Fanuc TP program (LS listing): hs_ov_h80_gutr1.ls

/PROG  hs_ov_h80_gutr1
/ATTR
COMMENT	= "19-03-05 13:35:50";
PROG_SIZE	= 0;
DEFAULT_GROUP	= 1, *, *, *, *;
/APPL
    ARC Welding Equipment: 1, *, *, *, *;
/MN
   1:  CALL HOME_ALL;
   1:  UFRAME_NUM = 1;
   1:  UTOOL_NUM = 3;
   1:  COL GUARD ADJUST 150;
   1:  PR[91] = PR[90];
   1:  PR[91,1] = PR[90,1] + -0.906;
   1:  PR[91,2] = PR[90,2] + 14.621;
   1:  PR[91,3] = PR[90,3] + 36.595;
   1:  PR[92] = PR[91];
   1:  PR[92,3] = PR[92,3] + 50;
   1:J PR[92] 10% FINE;
   1:L PR[91] R[100]mm/sec CNT100;
   1:  CALL LASER_DRAHT_START;
   1:  PR[91,1] = PR[90,1] + -1.737;
   1:  PR[91,2] = PR[90,2] + 15.006;
   1:L PR[91] R[100]mm/sec CNT100;
   1:  PR[91,1] = PR[90,1] + -2.132;
   1:  PR[91,2] = PR[90,2] + 15.132;
   1:L PR[91] R[100]mm/sec CNT100;
   1:  PR[91,1] = PR[90,1] + -6.402;
   1:  PR[91,2] = PR[90,2] + 17.485;
   1:L PR[91] R[100]mm/sec CNT100;
   1:  PR[91,1] = PR[90,1] + -10.845;
   1:  PR[91,2] = PR[90,2] + 18.832;
   1:L PR[91] R[100]mm/sec CNT100;
   1:  PR[91,1] = PR[90,1] + -10.901;
   1:  PR[91,2] = PR[90,2] + 18.841;
   1:L PR[91] R[100]mm/sec CNT100;
   1:  PR[91,1] = PR[90,1] + -15.199;
   1:  PR[91,2] = PR[90,2] + 19.185;
   1:L PR[91] R[100]mm/sec CNT100;
   1:  PR[91,1] = PR[90,1] + -15.522;
   1:  PR[91,2] = PR[90,2] + 19.196;
   1:L PR[91] R[100]mm/sec CNT100;
   1:  PR[91,1] = PR[90,1] + -15.935;
   1:  PR[91,2] = PR[90,2] + 19.155;
   1:L PR[91] R[100]mm/sec CNT100;
   1:  PR[91,1] = PR[90,1] + -19.834;
   1:  PR[91,2] = PR[90,2] + 18.637;
   1:L PR[91] R[100]mm/sec CNT100;
   1:  PR[91,1] = PR[90,1] + -20.377;
   1:  PR[91,2] = PR[90,2] + 18.508;
   1:L PR[91] R[100]mm/sec CNT100;
   1:  PR[91,1] = PR[90,1] + -21.139;
   1:  PR[91,2] = PR[90,2] + 18.219;
   1:L PR[91] R[100]mm/sec CNT100;
   1:  PR[91,1] = PR[90,1] + -24.417;
   1:  PR[91,2] = PR[90,2] + 17.039;
   1:L PR[91] R[100]mm/sec CNT100;
   1:  PR[91,1] = PR[90,1] + -25.209;
   1:  PR[91,2] = PR[90,2] + 16.607;
   1:L PR[91] R[100]mm/sec CNT100;
   1:  PR[91,1] = PR[90,1] + -27.740;
   1:  PR[91,2] = PR[90,2] + 15.030;
   1:L PR[91] R[100]mm/sec CNT100;
   1:  PR[91,1] = PR[90,1] + -28.583;
   1:  PR[91,2] = PR[90,2] + 14.408;
   1:L PR[91] R[100]mm/sec CNT100;
   1:  PR[91,1] = PR[90,1] + -31.305;
   1:  PR[91,2] = PR[90,2] + 11.747;
   1:L PR[91] R[100]mm/sec CNT100;
   1:  PR[91,1] = PR[90,1] + -32.081;
   1:  PR[91,2] = PR[90,2] + 10.737;
   1:L PR[91] R[100]mm/sec CNT100;
   1:  PR[91,1] = PR[90,1] + -33.285;
   1:  PR[91,2] = PR[90,2] + 8.860;
   1:L PR[91] R[100]mm/sec CNT100;
   1:  PR[91,1] = PR[90,1] + -33.988;
   1:  PR[91,2] = PR[90,2] + 7.608;
   1:L PR[91] R[100]mm/sec CNT100;
   1:  PR[91,1] = PR[90,1] + -34.555;
   1:  PR[91,2] = PR[90,2] + 6.149;
   1:L PR[91] R[100]mm/sec CNT100;
   1:  PR[91,1] = PR[90,1] + -35.218;
   1:  PR[91,2] = PR[90,2] + 4.337;
   1:L PR[91] R[100]mm/sec CNT100;
   1:  PR[91,1] = PR[90,1] + -35.516;
   1:  PR[91,2] = PR[90,2] + 3.007;
   1:L PR[91] R[100]mm/sec CNT100;
   1:  PR[91,1] = PR[90,1] + -35.629;
   1:  PR[91,2] = PR[90,2] + 1.384;
   1:L PR[91] R[100]mm/sec CNT100;
   1:  PR[91,1] = PR[90,1] + -35.844;
   1:  PR[91,2] = PR[90,2] + -0.479;
   1:L PR[91] R[100]mm/sec CNT100;
   1:  PR[91,1] = PR[90,1] + -35.742;
   1:  PR[91,2] = PR[90,2] + -1.958;
   1:L PR[91] R[100]mm/sec CNT100;
   1:  PR[91,1] = PR[90,1] + -35.528;
   1:  PR[91,2] = PR[90,2] + -3.801;
   1:L PR[91] R[100]mm/sec CNT100;
   1:  PR[91,1] = PR[90,1] + -35.224;
   1:  PR[91,2] = PR[90,2] + -5.160;
   1:L PR[91] R[100]mm/sec CNT100;
   1:  PR[91,1] = PR[90,1] + -34.654;
   1:  PR[91,2] = PR[90,2] + -6.622;
   1:L PR[91] R[100]mm/sec CNT100;
   1:  PR[91,1] = PR[90,1] + -33.976;
   1:  PR[91,2] = PR[90,2] + -8.476;
   1:L PR[91] R[100]mm/sec CNT100;
   1:  PR[91,1] = PR[90,1] + -33.285;
   1:  PR[91,2] = PR[90,2] + -9.707;
   1:L PR[91] R[100]mm/sec CNT100;
   1:  PR[91,1] = PR[90,1] + -32.081;
   1:  PR[91,2] = PR[90,2] + -11.584;
   1:L PR[91] R[100]mm/sec CNT100;
   1:  PR[91,1] = PR[90,1] + -31.305;
   1:  PR[91,2] = PR[90,2] + -12.594;
   1:L PR[91] R[100]mm/sec CNT100;
   1:  PR[91,1] = PR[90,1] + -28.583;
   1:  PR[91,2] = PR[90,2] + -15.255;
   1:L PR[91] R[100]mm/sec CNT100;
   1:  PR[91,1] = PR[90,1] + -27.740;
   1:  PR[91,2] = PR[90,2] + -15.877;
   1:L PR[91] R[100]mm/sec CNT100;
   1:  PR[91,1] = PR[90,1] + -25.208;
   1:  PR[91,2] = PR[90,2] + -17.454;
   1:L PR[91] R[100]mm/sec CNT100;
   1:  PR[91,1] = PR[90,1] + -24.396;
   1:  PR[91,2] = PR[90,2] + -17.898;
   1:L PR[91] R[100]mm/sec CNT100;
   1:  PR[91,1] = PR[90,1] + -23.616;
   1:  PR[91,2] = PR[90,2] + -18.195;
   1:L PR[91] R[100]mm/sec CNT100;
   1:  PR[91,1] = PR[90,1] + -20.398;
   1:  PR[91,2] = PR[90,2] + -19.351;
   1:L PR[91] R[100]mm/sec CNT100;
   1:  PR[91,1] = PR[90,1] + -19.877;
   1:  PR[91,2] = PR[90,2] + -19.474;
   1:L PR[91] R[100]mm/sec CNT100;
   1:  PR[91,1] = PR[90,1] + -19.263;
   1:  PR[91,2] = PR[90,2] + -19.533;
   1:L PR[91] R[100]mm/sec CNT100;
   1:  PR[91,1] = PR[90,1] + -15.479;
   1:  PR[91,2] = PR[90,2] + -20.042;
   1:L PR[91] R[100]mm/sec CNT100;
   1:  PR[91,1] = PR[90,1] + -15.199;
   1:  PR[91,2] = PR[90,2] + -20.033;
   1:L PR[91] R[100]mm/sec CNT100;
   1:  PR[91,1] = PR[90,1] + -10.901;
   1:  PR[91,2] = PR[90,2] + -19.688;
   1:L PR[91] R[100]mm/sec CNT100;
   1:  PR[91,1] = PR[90,1] + -10.845;
   1:  PR[91,2] = PR[90,2] + -19.679;
   1:L PR[91] R[100]mm/sec CNT100;
   1:  PR[91,1] = PR[90,1] + -6.401;
   1:  PR[91,2] = PR[90,2] + -18.332;
   1:L PR[91] R[100]mm/sec CNT100;
   1:  PR[91,1] = PR[90,1] + -2.136;
   1:  PR[91,2] = PR[90,2] + -15.981;
   1:L PR[91] R[100]mm/sec CNT100;
   1:  PR[91,1] = PR[90,1] + -1.638;
   1:  PR[91,2] = PR[90,2] + -15.821;
   1:L PR[91] R[100]mm/sec CNT100;
   1:  PR[91,1] = PR[90,1] + -1.622;
   1:  PR[91,2] = PR[90,2] + -15.815;
   1:L PR[91] R[100]mm/sec CNT100;
   1:  PR[91,1] = PR[90,1] + -0.788;
   1:  PR[91,2] = PR[90,2] + -15.263;
   1:L PR[91] R[100]mm/sec CNT100;
   1:  PR[91,1] = PR[90,1] + 0.384;
   1:  PR[91,2] = PR[90,2] + -15.590;
   1:L PR[91] R[100]mm/sec CNT100;
   1:  PR[91,1] = PR[90,1] + 1.398;
   1:  PR[91,2] = PR[90,2] + -15.747;
   1:L PR[91] R[100]mm/sec CNT100;
   1:  PR[91,1] = PR[90,1] + 1.978;
   1:  PR[91,2] = PR[90,2] + -16.161;
   1:L PR[91] R[100]mm/sec CNT100;
   1:  PR[91,1] = PR[90,1] + 5.916;
   1:  PR[91,2] = PR[90,2] + -18.330;
   1:L PR[91] R[100]mm/sec CNT100;
   1:  PR[91,1] = PR[90,1] + 10.362;
   1:  PR[91,2] = PR[90,2] + -19.678;
   1:L PR[91] R[100]mm/sec CNT100;
   1:  PR[91,1] = PR[90,1] + 10.418;
   1:  PR[91,2] = PR[90,2] + -19.687;
   1:L PR[91] R[100]mm/sec CNT100;
   1:  PR[91,1] = PR[90,1] + 14.716;
   1:  PR[91,2] = PR[90,2] + -20.033;
   1:L PR[91] R[100]mm/sec CNT100;
   1:  PR[91,1] = PR[90,1] + 15.037;
   1:  PR[91,2] = PR[90,2] + -20.044;
   1:L PR[91] R[100]mm/sec CNT100;
   1:  PR[91,1] = PR[90,1] + 15.446;
   1:  PR[91,2] = PR[90,2] + -20.004;
   1:L PR[91] R[100]mm/sec CNT100;
   1:  PR[91,1] = PR[90,1] + 19.345;
   1:  PR[91,2] = PR[90,2] + -19.485;
   1:L PR[91] R[100]mm/sec CNT100;
   1:  PR[91,1] = PR[90,1] + 19.888;
   1:  PR[91,2] = PR[90,2] + -19.357;
   1:L PR[91] R[100]mm/sec CNT100;
   1:  PR[91,1] = PR[90,1] + 20.651;
   1:  PR[91,2] = PR[90,2] + -19.069;
   1:L PR[91] R[100]mm/sec CNT100;
   1:  PR[91,1] = PR[90,1] + 23.931;
   1:  PR[91,2] = PR[90,2] + -17.890;
   1:L PR[91] R[100]mm/sec CNT100;
   1:  PR[91,1] = PR[90,1] + 24.719;
   1:  PR[91,2] = PR[90,2] + -17.462;
   1:L PR[91] R[100]mm/sec CNT100;
   1:  PR[91,1] = PR[90,1] + 27.251;
   1:  PR[91,2] = PR[90,2] + -15.887;
   1:L PR[91] R[100]mm/sec CNT100;
   1:  PR[91,1] = PR[90,1] + 28.082;
   1:  PR[91,2] = PR[90,2] + -15.277;
   1:L PR[91] R[100]mm/sec CNT100;
   1:  PR[91,1] = PR[90,1] + 30.802;
   1:  PR[91,2] = PR[90,2] + -12.615;
   1:L PR[91] R[100]mm/sec CNT100;
   1:  PR[91,1] = PR[90,1] + 31.587;
   1:  PR[91,2] = PR[90,2] + -11.595;
   1:L PR[91] R[100]mm/sec CNT100;
   1:  PR[91,1] = PR[90,1] + 32.794;
   1:  PR[91,2] = PR[90,2] + -9.717;
   1:L PR[91] R[100]mm/sec CNT100;
   1:  PR[91,1] = PR[90,1] + 33.504;
   1:  PR[91,2] = PR[90,2] + -8.463;
   1:L PR[91] R[100]mm/sec CNT100;
   1:  PR[91,1] = PR[90,1] + 34.067;
   1:  PR[91,2] = PR[90,2] + -7.036;
   1:L PR[91] R[100]mm/sec CNT100;
   1:  PR[91,1] = PR[90,1] + 34.729;
   1:  PR[91,2] = PR[90,2] + -5.233;
   1:L PR[91] R[100]mm/sec CNT100;
   1:  PR[91,1] = PR[90,1] + 35.030;
   1:  PR[91,2] = PR[90,2] + -3.913;
   1:L PR[91] R[100]mm/sec CNT100;
   1:  PR[91,1] = PR[90,1] + 35.150;
   1:  PR[91,2] = PR[90,2] + -2.237;
   1:L PR[91] R[100]mm/sec CNT100;
   1:  PR[91,1] = PR[90,1] + 35.364;
   1:  PR[91,2] = PR[90,2] + -0.371;
   1:L PR[91] R[100]mm/sec CNT100;
   1:  PR[91,1] = PR[90,1] + 35.255;
   1:  PR[91,2] = PR[90,2] + 1.165;
   1:L PR[91] R[100]mm/sec CNT100;
   1:  PR[91,1] = PR[90,1] + 35.042;
   1:  PR[91,2] = PR[90,2] + 3.015;
   1:L PR[91] R[100]mm/sec CNT100;
   1:  PR[91,1] = PR[90,1] + 34.736;
   1:  PR[91,2] = PR[90,2] + 4.358;
   1:L PR[91] R[100]mm/sec CNT100;
   1:  PR[91,1] = PR[90,1] + 34.169;
   1:  PR[91,2] = PR[90,2] + 5.793;
   1:L PR[91] R[100]mm/sec CNT100;
   1:  PR[91,1] = PR[90,1] + 33.490;
   1:  PR[91,2] = PR[90,2] + 7.640;
   1:L PR[91] R[100]mm/sec CNT100;
   1:  PR[91,1] = PR[90,1] + 32.794;
   1:  PR[91,2] = PR[90,2] + 8.870;
   1:L PR[91] R[100]mm/sec CNT100;
   1:  PR[91,1] = PR[90,1] + 31.587;
   1:  PR[91,2] = PR[90,2] + 10.747;
   1:L PR[91] R[100]mm/sec CNT100;
   1:  PR[91,1] = PR[90,1] + 30.802;
   1:  PR[91,2] = PR[90,2] + 11.767;
   1:L PR[91] R[100]mm/sec CNT100;
   1:  PR[91,1] = PR[90,1] + 28.082;
   1:  PR[91,2] = PR[90,2] + 14.429;
   1:L PR[91] R[100]mm/sec CNT100;
   1:  PR[91,1] = PR[90,1] + 27.251;
   1:  PR[91,2] = PR[90,2] + 15.039;
   1:L PR[91] R[100]mm/sec CNT100;
   1:  PR[91,1] = PR[90,1] + 24.719;
   1:  PR[91,2] = PR[90,2] + 16.614;
   1:L PR[91] R[100]mm/sec CNT100;
   1:  PR[91,1] = PR[90,1] + 23.912;
   1:  PR[91,2] = PR[90,2] + 17.052;
   1:L PR[91] R[100]mm/sec CNT100;
   1:  PR[91,1] = PR[90,1] + 23.128;
   1:  PR[91,2] = PR[90,2] + 17.350;
   1:L PR[91] R[100]mm/sec CNT100;
   1:  PR[91,1] = PR[90,1] + 19.908;
   1:  PR[91,2] = PR[90,2] + 18.505;
   1:L PR[91] R[100]mm/sec CNT100;
   1:  PR[91,1] = PR[90,1] + 19.390;
   1:  PR[91,2] = PR[90,2] + 18.628;
   1:L PR[91] R[100]mm/sec CNT100;
   1:  PR[91,1] = PR[90,1] + 18.778;
   1:  PR[91,2] = PR[90,2] + 18.685;
   1:L PR[91] R[100]mm/sec CNT100;
   1:  PR[91,1] = PR[90,1] + 14.994;
   1:  PR[91,2] = PR[90,2] + 19.195;
   1:L PR[91] R[100]mm/sec CNT100;
   1:  PR[91,1] = PR[90,1] + 14.716;
   1:  PR[91,2] = PR[90,2] + 19.186;
   1:L PR[91] R[100]mm/sec CNT100;
   1:  PR[91,1] = PR[90,1] + 10.418;
   1:  PR[91,2] = PR[90,2] + 18.840;
   1:L PR[91] R[100]mm/sec CNT100;
   1:  PR[91,1] = PR[90,1] + 10.362;
   1:  PR[91,2] = PR[90,2] + 18.830;
   1:L PR[91] R[100]mm/sec CNT100;
   1:  PR[91,1] = PR[90,1] + 5.916;
   1:  PR[91,2] = PR[90,2] + 17.483;
   1:L PR[91] R[100]mm/sec CNT100;
   1:  PR[91,1] = PR[90,1] + 1.978;
   1:  PR[91,2] = PR[90,2] + 15.314;
   1:L PR[91] R[100]mm/sec CNT100;
   1:  PR[91,1] = PR[90,1] + 1.394;
   1:  PR[91,2] = PR[90,2] + 14.896;
   1:L PR[91] R[100]mm/sec CNT100;
   1:  PR[91,1] = PR[90,1] + 0.531;
   1:  PR[91,2] = PR[90,2] + 14.765;
   1:L PR[91] R[100]mm/sec CNT100;
   1:  PR[91,1] = PR[90,1] + 0.191;
   1:  PR[91,2] = PR[90,2] + 14.622;
   1:L PR[91] R[100]mm/sec CNT100;
   1:  PR[91] = PR[90];
   1:  PR[91,1] = PR[90,1] + -2.097;
   1:  PR[91,2] = PR[90,2] + 15.618;
   1:  PR[91,3] = PR[90,3] + 37.895;
   1:L PR[91] R[100]mm/sec CNT100;
   1:  PR[91,1] = PR[90,1] + -5.253;
   1:  PR[91,2] = PR[90,2] + 17.345;
   1:L PR[91] R[100]mm/sec CNT100;
   1:  PR[91,1] = PR[90,1] + -5.848;
   1:  PR[91,2] = PR[90,2] + 17.646;
   1:L PR[91] R[100]mm/sec CNT100;
   1:  PR[91,1] = PR[90,1] + -10.319;
   1:  PR[91,2] = PR[90,2] + 18.953;
   1:L PR[91] R[100]mm/sec CNT100;
   1:  PR[91,1] = PR[90,1] + -15.016;
   1:  PR[91,2] = PR[90,2] + 19.315;
   1:L PR[91] R[100]mm/sec CNT100;
   1:  PR[91,1] = PR[90,1] + -19.530;
   1:  PR[91,2] = PR[90,2] + 18.722;
   1:L PR[91] R[100]mm/sec CNT100;
   1:  PR[91,1] = PR[90,1] + -19.752;
   1:  PR[91,2] = PR[90,2] + 18.670;
   1:L PR[91] R[100]mm/sec CNT100;
   1:  PR[91,1] = PR[90,1] + -23.990;
   1:  PR[91,2] = PR[90,2] + 17.135;
   1:L PR[91] R[100]mm/sec CNT100;
   1:  PR[91,1] = PR[90,1] + -24.457;
   1:  PR[91,2] = PR[90,2] + 16.880;
   1:L PR[91] R[100]mm/sec CNT100;
   1:  PR[91,1] = PR[90,1] + -27.491;
   1:  PR[91,2] = PR[90,2] + 14.990;
   1:L PR[91] R[100]mm/sec CNT100;
   1:  PR[91,1] = PR[90,1] + -28.052;
   1:  PR[91,2] = PR[90,2] + 14.576;
   1:L PR[91] R[100]mm/sec CNT100;
   1:  PR[91,1] = PR[90,1] + -30.941;
   1:  PR[91,2] = PR[90,2] + 11.749;
   1:L PR[91] R[100]mm/sec CNT100;
   1:  PR[91,1] = PR[90,1] + -31.495;
   1:  PR[91,2] = PR[90,2] + 11.027;
   1:L PR[91] R[100]mm/sec CNT100;
   1:  PR[91,1] = PR[90,1] + -33.019;
   1:  PR[91,2] = PR[90,2] + 8.652;
   1:L PR[91] R[100]mm/sec CNT100;
   1:  PR[91,1] = PR[90,1] + -33.545;
   1:  PR[91,2] = PR[90,2] + 7.714;
   1:L PR[91] R[100]mm/sec CNT100;
   1:  PR[91,1] = PR[90,1] + -33.976;
   1:  PR[91,2] = PR[90,2] + 6.608;
   1:L PR[91] R[100]mm/sec CNT100;
   1:  PR[91,1] = PR[90,1] + -34.843;
   1:  PR[91,2] = PR[90,2] + 4.238;
   1:L PR[91] R[100]mm/sec CNT100;
   1:  PR[91,1] = PR[90,1] + -35.065;
   1:  PR[91,2] = PR[90,2] + 3.248;
   1:L PR[91] R[100]mm/sec CNT100;
   1:  PR[91,1] = PR[90,1] + -35.153;
   1:  PR[91,2] = PR[90,2] + 1.982;
   1:L PR[91] R[100]mm/sec CNT100;
   1:  PR[91,1] = PR[90,1] + -35.437;
   1:  PR[91,2] = PR[90,2] + -0.479;
   1:L PR[91] R[100]mm/sec CNT100;
   1:  PR[91,1] = PR[90,1] + -35.359;
   1:  PR[91,2] = PR[90,2] + -1.608;
   1:L PR[91] R[100]mm/sec CNT100;
   1:  PR[91,1] = PR[90,1] + -35.077;
   1:  PR[91,2] = PR[90,2] + -4.042;
   1:L PR[91] R[100]mm/sec CNT100;
   1:  PR[91,1] = PR[90,1] + -34.849;
   1:  PR[91,2] = PR[90,2] + -5.061;
   1:L PR[91] R[100]mm/sec CNT100;
   1:  PR[91,1] = PR[90,1] + -34.407;
   1:  PR[91,2] = PR[90,2] + -6.195;
   1:L PR[91] R[100]mm/sec CNT100;
   1:  PR[91,1] = PR[90,1] + -33.533;
   1:  PR[91,2] = PR[90,2] + -8.583;
   1:L PR[91] R[100]mm/sec CNT100;
   1:  PR[91,1] = PR[90,1] + -33.019;
   1:  PR[91,2] = PR[90,2] + -9.499;
   1:L PR[91] R[100]mm/sec CNT100;
   1:  PR[91,1] = PR[90,1] + -31.495;
   1:  PR[91,2] = PR[90,2] + -11.874;
   1:L PR[91] R[100]mm/sec CNT100;
   1:  PR[91,1] = PR[90,1] + -30.941;
   1:  PR[91,2] = PR[90,2] + -12.597;
   1:L PR[91] R[100]mm/sec CNT100;
   1:  PR[91,1] = PR[90,1] + -28.051;
   1:  PR[91,2] = PR[90,2] + -15.424;
   1:L PR[91] R[100]mm/sec CNT100;
   1:  PR[91,1] = PR[90,1] + -27.491;
   1:  PR[91,2] = PR[90,2] + -15.837;
   1:L PR[91] R[100]mm/sec CNT100;
   1:  PR[91,1] = PR[90,1] + -24.457;
   1:  PR[91,2] = PR[90,2] + -17.727;
   1:L PR[91] R[100]mm/sec CNT100;
   1:  PR[91,1] = PR[90,1] + -23.971;
   1:  PR[91,2] = PR[90,2] + -17.992;
   1:L PR[91] R[100]mm/sec CNT100;
   1:  PR[91,1] = PR[90,1] + -23.498;
   1:  PR[91,2] = PR[90,2] + -18.173;
   1:L PR[91] R[100]mm/sec CNT100;
   1:  PR[91,1] = PR[90,1] + -19.755;
   1:  PR[91,2] = PR[90,2] + -19.516;
   1:L PR[91] R[100]mm/sec CNT100;
   1:  PR[91,1] = PR[90,1] + -19.571;
   1:  PR[91,2] = PR[90,2] + -19.560;
   1:L PR[91] R[100]mm/sec CNT100;
   1:  PR[91,1] = PR[90,1] + -19.261;
   1:  PR[91,2] = PR[90,2] + -19.590;
   1:L PR[91] R[100]mm/sec CNT100;
   1:  PR[91,1] = PR[90,1] + -15.011;
   1:  PR[91,2] = PR[90,2] + -20.162;
   1:L PR[91] R[100]mm/sec CNT100;
   1:  PR[91,1] = PR[90,1] + -10.319;
   1:  PR[91,2] = PR[90,2] + -19.800;
   1:L PR[91] R[100]mm/sec CNT100;
   1:  PR[91,1] = PR[90,1] + -5.848;
   1:  PR[91,2] = PR[90,2] + -18.493;
   1:L PR[91] R[100]mm/sec CNT100;
   1:  PR[91,1] = PR[90,1] + -5.233;
   1:  PR[91,2] = PR[90,2] + -18.182;
   1:L PR[91] R[100]mm/sec CNT100;
   1:  PR[91,1] = PR[90,1] + -2.098;
   1:  PR[91,2] = PR[90,2] + -16.466;
   1:L PR[91] R[100]mm/sec CNT100;
   1:  PR[91,1] = PR[90,1] + -0.302;
   1:  PR[91,2] = PR[90,2] + -15.887;
   1:L PR[91] R[100]mm/sec CNT100;
   1:  PR[91,1] = PR[90,1] + 0.369;
   1:  PR[91,2] = PR[90,2] + -16.121;
   1:L PR[91] R[100]mm/sec CNT100;
   1:  PR[91,1] = PR[90,1] + 1.439;
   1:  PR[91,2] = PR[90,2] + -16.285;
   1:L PR[91] R[100]mm/sec CNT100;
   1:  PR[91,1] = PR[90,1] + 1.941;
   1:  PR[91,2] = PR[90,2] + -16.645;
   1:L PR[91] R[100]mm/sec CNT100;
   1:  PR[91,1] = PR[90,1] + 4.765;
   1:  PR[91,2] = PR[90,2] + -18.189;
   1:L PR[91] R[100]mm/sec CNT100;
   1:  PR[91,1] = PR[90,1] + 5.363;
   1:  PR[91,2] = PR[90,2] + -18.491;
   1:L PR[91] R[100]mm/sec CNT100;
   1:  PR[91,1] = PR[90,1] + 9.835;
   1:  PR[91,2] = PR[90,2] + -19.798;
   1:L PR[91] R[100]mm/sec CNT100;
   1:  PR[91,1] = PR[90,1] + 14.531;
   1:  PR[91,2] = PR[90,2] + -20.162;
   1:L PR[91] R[100]mm/sec CNT100;
   1:  PR[91,1] = PR[90,1] + 19.044;
   1:  PR[91,2] = PR[90,2] + -19.570;
   1:L PR[91] R[100]mm/sec CNT100;
   1:  PR[91,1] = PR[90,1] + 19.265;
   1:  PR[91,2] = PR[90,2] + -19.518;
   1:L PR[91] R[100]mm/sec CNT100;
   1:  PR[91,1] = PR[90,1] + 23.506;
   1:  PR[91,2] = PR[90,2] + -17.984;
   1:L PR[91] R[100]mm/sec CNT100;
   1:  PR[91,1] = PR[90,1] + 23.971;
   1:  PR[91,2] = PR[90,2] + -17.732;
   1:L PR[91] R[100]mm/sec CNT100;
   1:  PR[91,1] = PR[90,1] + 27.004;
   1:  PR[91,2] = PR[90,2] + -15.845;
   1:L PR[91] R[100]mm/sec CNT100;
   1:  PR[91,1] = PR[90,1] + 27.556;
   1:  PR[91,2] = PR[90,2] + -15.440;
   1:L PR[91] R[100]mm/sec CNT100;
   1:  PR[91,1] = PR[90,1] + 30.443;
   1:  PR[91,2] = PR[90,2] + -12.611;
   1:L PR[91] R[100]mm/sec CNT100;
   1:  PR[91,1] = PR[90,1] + 31.005;
   1:  PR[91,2] = PR[90,2] + -11.881;
   1:L PR[91] R[100]mm/sec CNT100;
   1:  PR[91,1] = PR[90,1] + 32.531;
   1:  PR[91,2] = PR[90,2] + -9.506;
   1:L PR[91] R[100]mm/sec CNT100;
   1:  PR[91,1] = PR[90,1] + 33.064;
   1:  PR[91,2] = PR[90,2] + -8.566;
   1:L PR[91] R[100]mm/sec CNT100;
   1:  PR[91,1] = PR[90,1] + 33.490;
   1:  PR[91,2] = PR[90,2] + -7.485;
   1:L PR[91] R[100]mm/sec CNT100;
   1:  PR[91,1] = PR[90,1] + 34.356;
   1:  PR[91,2] = PR[90,2] + -5.127;
   1:L PR[91] R[100]mm/sec CNT100;
   1:  PR[91,1] = PR[90,1] + 34.580;
   1:  PR[91,2] = PR[90,2] + -4.145;
   1:L PR[91] R[100]mm/sec CNT100;
   1:  PR[91,1] = PR[90,1] + 34.673;
   1:  PR[91,2] = PR[90,2] + -2.838;
   1:L PR[91] R[100]mm/sec CNT100;
   1:  PR[91,1] = PR[90,1] + 34.957;
   1:  PR[91,2] = PR[90,2] + -0.371;
   1:L PR[91] R[100]mm/sec CNT100;
   1:  PR[91,1] = PR[90,1] + 34.874;
   1:  PR[91,2] = PR[90,2] + 0.804;
   1:L PR[91] R[100]mm/sec CNT100;
   1:  PR[91,1] = PR[90,1] + 34.592;
   1:  PR[91,2] = PR[90,2] + 3.246;
   1:L PR[91] R[100]mm/sec CNT100;
   1:  PR[91,1] = PR[90,1] + 34.363;
   1:  PR[91,2] = PR[90,2] + 4.252;
   1:L PR[91] R[100]mm/sec CNT100;
   1:  PR[91,1] = PR[90,1] + 33.923;
   1:  PR[91,2] = PR[90,2] + 5.364;
   1:L PR[91] R[100]mm/sec CNT100;
   1:  PR[91,1] = PR[90,1] + 33.050;
   1:  PR[91,2] = PR[90,2] + 7.743;
   1:L PR[91] R[100]mm/sec CNT100;
   1:  PR[91,1] = PR[90,1] + 32.531;
   1:  PR[91,2] = PR[90,2] + 8.659;
   1:L PR[91] R[100]mm/sec CNT100;
   1:  PR[91,1] = PR[90,1] + 31.005;
   1:  PR[91,2] = PR[90,2] + 11.033;
   1:L PR[91] R[100]mm/sec CNT100;
   1:  PR[91,1] = PR[90,1] + 30.443;
   1:  PR[91,2] = PR[90,2] + 11.764;
   1:L PR[91] R[100]mm/sec CNT100;
   1:  PR[91,1] = PR[90,1] + 27.556;
   1:  PR[91,2] = PR[90,2] + 14.593;
   1:L PR[91] R[100]mm/sec CNT100;
   1:  PR[91,1] = PR[90,1] + 27.004;
   1:  PR[91,2] = PR[90,2] + 14.998;
   1:L PR[91] R[100]mm/sec CNT100;
   1:  PR[91,1] = PR[90,1] + 23.971;
   1:  PR[91,2] = PR[90,2] + 16.885;
   1:L PR[91] R[100]mm/sec CNT100;
   1:  PR[91,1] = PR[90,1] + 23.489;
   1:  PR[91,2] = PR[90,2] + 17.146;
   1:L PR[91] R[100]mm/sec CNT100;
   1:  PR[91,1] = PR[90,1] + 23.013;
   1:  PR[91,2] = PR[90,2] + 17.327;
   1:L PR[91] R[100]mm/sec CNT100;
   1:  PR[91,1] = PR[90,1] + 19.268;
   1:  PR[91,2] = PR[90,2] + 18.670;
   1:L PR[91] R[100]mm/sec CNT100;
   1:  PR[91,1] = PR[90,1] + 19.087;
   1:  PR[91,2] = PR[90,2] + 18.713;
   1:L PR[91] R[100]mm/sec CNT100;
   1:  PR[91,1] = PR[90,1] + 18.778;
   1:  PR[91,2] = PR[90,2] + 18.742;
   1:L PR[91] R[100]mm/sec CNT100;
   1:  PR[91,1] = PR[90,1] + 14.527;
   1:  PR[91,2] = PR[90,2] + 19.315;
   1:L PR[91] R[100]mm/sec CNT100;
   1:  PR[91,1] = PR[90,1] + 9.836;
   1:  PR[91,2] = PR[90,2] + 18.951;
   1:L PR[91] R[100]mm/sec CNT100;
   1:  PR[91,1] = PR[90,1] + 5.363;
   1:  PR[91,2] = PR[90,2] + 17.644;
   1:L PR[91] R[100]mm/sec CNT100;
   1:  PR[91,1] = PR[90,1] + 4.771;
   1:  PR[91,2] = PR[90,2] + 17.345;
   1:L PR[91] R[100]mm/sec CNT100;
   1:  PR[91,1] = PR[90,1] + 1.938;
   1:  PR[91,2] = PR[90,2] + 15.796;
   1:L PR[91] R[100]mm/sec CNT100;
   1:  PR[91,1] = PR[90,1] + 1.434;
   1:  PR[91,2] = PR[90,2] + 15.436;
   1:L PR[91] R[100]mm/sec CNT100;
   1:  PR[91,1] = PR[90,1] + 0.367;
   1:  PR[91,2] = PR[90,2] + 15.273;
   1:L PR[91] R[100]mm/sec CNT100;
   1:  PR[91,1] = PR[90,1] + -0.302;
   1:  PR[91,2] = PR[90,2] + 15.040;
   1:L PR[91] R[100]mm/sec CNT100;
   1:  PR[91] = PR[90];
   1:  PR[91,1] = PR[90,1] + -2.076;
   1:  PR[91,2] = PR[90,2] + 16.111;
   1:  PR[91,3] = PR[90,3] + 39.195;
   1:L PR[91] R[100]mm/sec CNT100;
   1:  PR[91,1] = PR[90,1] + -3.718;
   1:  PR[91,2] = PR[90,2] + 17.010;
   1:L PR[91] R[100]mm/sec CNT100;
   1:  PR[91,1] = PR[90,1] + -5.377;
   1:  PR[91,2] = PR[90,2] + 17.850;
   1:L PR[91] R[100]mm/sec CNT100;
   1:  PR[91,1] = PR[90,1] + -9.457;
   1:  PR[91,2] = PR[90,2] + 19.043;
   1:L PR[91] R[100]mm/sec CNT100;
   1:  PR[91,1] = PR[90,1] + -9.837;
   1:  PR[91,2] = PR[90,2] + 19.143;
   1:L PR[91] R[100]mm/sec CNT100;
   1:  PR[91,1] = PR[90,1] + -14.504;
   1:  PR[91,2] = PR[90,2] + 19.459;
   1:L PR[91] R[100]mm/sec CNT100;
   1:  PR[91,1] = PR[90,1] + -16.542;
   1:  PR[91,2] = PR[90,2] + 19.165;
   1:L PR[91] R[100]mm/sec CNT100;
   1:  PR[91,1] = PR[90,1] + -19.162;
   1:  PR[91,2] = PR[90,2] + 18.817;
   1:L PR[91] R[100]mm/sec CNT100;
   1:  PR[91,1] = PR[90,1] + -23.567;
   1:  PR[91,2] = PR[90,2] + 17.229;
   1:L PR[91] R[100]mm/sec CNT100;
   1:  PR[91,1] = PR[90,1] + -23.706;
   1:  PR[91,2] = PR[90,2] + 17.153;
   1:L PR[91] R[100]mm/sec CNT100;
   1:  PR[91,1] = PR[90,1] + -27.242;
   1:  PR[91,2] = PR[90,2] + 14.950;
   1:L PR[91] R[100]mm/sec CNT100;
   1:  PR[91,1] = PR[90,1] + -27.520;
   1:  PR[91,2] = PR[90,2] + 14.745;
   1:L PR[91] R[100]mm/sec CNT100;
   1:  PR[91,1] = PR[90,1] + -30.576;
   1:  PR[91,2] = PR[90,2] + 11.752;
   1:L PR[91] R[100]mm/sec CNT100;
   1:  PR[91,1] = PR[90,1] + -30.910;
   1:  PR[91,2] = PR[90,2] + 11.317;
   1:L PR[91] R[100]mm/sec CNT100;
   1:  PR[91,1] = PR[90,1] + -32.753;
   1:  PR[91,2] = PR[90,2] + 8.444;
   1:L PR[91] R[100]mm/sec CNT100;
   1:  PR[91,1] = PR[90,1] + -33.103;
   1:  PR[91,2] = PR[90,2] + 7.821;
   1:L PR[91] R[100]mm/sec CNT100;
   1:  PR[91,1] = PR[90,1] + -33.396;
   1:  PR[91,2] = PR[90,2] + 7.067;
   1:L PR[91] R[100]mm/sec CNT100;
   1:  PR[91,1] = PR[90,1] + -34.468;
   1:  PR[91,2] = PR[90,2] + 4.139;
   1:L PR[91] R[100]mm/sec CNT100;
   1:  PR[91,1] = PR[90,1] + -34.614;
   1:  PR[91,2] = PR[90,2] + 3.489;
   1:L PR[91] R[100]mm/sec CNT100;
   1:  PR[91,1] = PR[90,1] + -34.677;
   1:  PR[91,2] = PR[90,2] + 2.581;
   1:L PR[91] R[100]mm/sec CNT100;
   1:  PR[91,1] = PR[90,1] + -35.030;
   1:  PR[91,2] = PR[90,2] + -0.479;
   1:L PR[91] R[100]mm/sec CNT100;
   1:  PR[91,1] = PR[90,1] + -34.976;
   1:  PR[91,2] = PR[90,2] + -1.258;
   1:L PR[91] R[100]mm/sec CNT100;
   1:  PR[91,1] = PR[90,1] + -34.626;
   1:  PR[91,2] = PR[90,2] + -4.282;
   1:L PR[91] R[100]mm/sec CNT100;
   1:  PR[91,1] = PR[90,1] + -34.473;
   1:  PR[91,2] = PR[90,2] + -4.962;
   1:L PR[91] R[100]mm/sec CNT100;
   1:  PR[91,1] = PR[90,1] + -34.160;
   1:  PR[91,2] = PR[90,2] + -5.767;
   1:L PR[91] R[100]mm/sec CNT100;
   1:  PR[91,1] = PR[90,1] + -33.091;
   1:  PR[91,2] = PR[90,2] + -8.690;
   1:L PR[91] R[100]mm/sec CNT100;
   1:  PR[91,1] = PR[90,1] + -32.753;
   1:  PR[91,2] = PR[90,2] + -9.292;
   1:L PR[91] R[100]mm/sec CNT100;
   1:  PR[91,1] = PR[90,1] + -30.910;
   1:  PR[91,2] = PR[90,2] + -12.164;
   1:L PR[91] R[100]mm/sec CNT100;
   1:  PR[91,1] = PR[90,1] + -30.576;
   1:  PR[91,2] = PR[90,2] + -12.599;
   1:L PR[91] R[100]mm/sec CNT100;
   1:  PR[91,1] = PR[90,1] + -27.520;
   1:  PR[91,2] = PR[90,2] + -15.592;
   1:L PR[91] R[100]mm/sec CNT100;
   1:  PR[91,1] = PR[90,1] + -27.242;
   1:  PR[91,2] = PR[90,2] + -15.797;
   1:L PR[91] R[100]mm/sec CNT100;
   1:  PR[91,1] = PR[90,1] + -23.706;
   1:  PR[91,2] = PR[90,2] + -18.000;
   1:L PR[91] R[100]mm/sec CNT100;
   1:  PR[91,1] = PR[90,1] + -23.566;
   1:  PR[91,2] = PR[90,2] + -18.076;
   1:L PR[91] R[100]mm/sec CNT100;
   1:  PR[91,1] = PR[90,1] + -19.162;
   1:  PR[91,2] = PR[90,2] + -19.664;
   1:L PR[91] R[100]mm/sec CNT100;
   1:  PR[91,1] = PR[90,1] + -16.543;
   1:  PR[91,2] = PR[90,2] + -20.012;
   1:L PR[91] R[100]mm/sec CNT100;
   1:  PR[91,1] = PR[90,1] + -14.503;
   1:  PR[91,2] = PR[90,2] + -20.307;
   1:L PR[91] R[100]mm/sec CNT100;
   1:  PR[91,1] = PR[90,1] + -9.836;
   1:  PR[91,2] = PR[90,2] + -19.990;
   1:L PR[91] R[100]mm/sec CNT100;
   1:  PR[91,1] = PR[90,1] + -9.456;
   1:  PR[91,2] = PR[90,2] + -19.890;
   1:L PR[91] R[100]mm/sec CNT100;
   1:  PR[91,1] = PR[90,1] + -5.329;
   1:  PR[91,2] = PR[90,2] + -18.683;
   1:L PR[91] R[100]mm/sec CNT100;
   1:  PR[91,1] = PR[90,1] + -5.307;
   1:  PR[91,2] = PR[90,2] + -18.673;
   1:L PR[91] R[100]mm/sec CNT100;
   1:  PR[91,1] = PR[90,1] + -3.680;
   1:  PR[91,2] = PR[90,2] + -17.837;
   1:L PR[91] R[100]mm/sec CNT100;
   1:  PR[91,1] = PR[90,1] + -2.077;
   1:  PR[91,2] = PR[90,2] + -16.960;
   1:L PR[91] R[100]mm/sec CNT100;
   1:  PR[91,1] = PR[90,1] + -0.280;
   1:  PR[91,2] = PR[90,2] + -16.350;
   1:L PR[91] R[100]mm/sec CNT100;
   1:  PR[91,1] = PR[90,1] + 0.770;
   1:  PR[91,2] = PR[90,2] + -16.716;
   1:L PR[91] R[100]mm/sec CNT100;
   1:  PR[91,1] = PR[90,1] + 1.485;
   1:  PR[91,2] = PR[90,2] + -16.825;
   1:L PR[91] R[100]mm/sec CNT100;
   1:  PR[91,1] = PR[90,1] + 1.908;
   1:  PR[91,2] = PR[90,2] + -17.132;
   1:L PR[91] R[100]mm/sec CNT100;
   1:  PR[91,1] = PR[90,1] + 3.235;
   1:  PR[91,2] = PR[90,2] + -17.857;
   1:L PR[91] R[100]mm/sec CNT100;
   1:  PR[91,1] = PR[90,1] + 4.821;
   1:  PR[91,2] = PR[90,2] + -18.670;
   1:L PR[91] R[100]mm/sec CNT100;
   1:  PR[91,1] = PR[90,1] + 4.845;
   1:  PR[91,2] = PR[90,2] + -18.681;
   1:L PR[91] R[100]mm/sec CNT100;
   1:  PR[91,1] = PR[90,1] + 8.973;
   1:  PR[91,2] = PR[90,2] + -19.889;
   1:L PR[91] R[100]mm/sec CNT100;
   1:  PR[91,1] = PR[90,1] + 9.353;
   1:  PR[91,2] = PR[90,2] + -19.988;
   1:L PR[91] R[100]mm/sec CNT100;
   1:  PR[91,1] = PR[90,1] + 14.020;
   1:  PR[91,2] = PR[90,2] + -20.307;
   1:L PR[91] R[100]mm/sec CNT100;
   1:  PR[91,1] = PR[90,1] + 16.062;
   1:  PR[91,2] = PR[90,2] + -20.012;
   1:L PR[91] R[100]mm/sec CNT100;
   1:  PR[91,1] = PR[90,1] + 18.678;
   1:  PR[91,2] = PR[90,2] + -19.664;
   1:L PR[91] R[100]mm/sec CNT100;
   1:  PR[91,1] = PR[90,1] + 23.085;
   1:  PR[91,2] = PR[90,2] + -18.077;
   1:L PR[91] R[100]mm/sec CNT100;
   1:  PR[91,1] = PR[90,1] + 23.223;
   1:  PR[91,2] = PR[90,2] + -18.002;
   1:L PR[91] R[100]mm/sec CNT100;
   1:  PR[91,1] = PR[90,1] + 26.758;
   1:  PR[91,2] = PR[90,2] + -15.803;
   1:L PR[91] R[100]mm/sec CNT100;
   1:  PR[91,1] = PR[90,1] + 27.029;
   1:  PR[91,2] = PR[90,2] + -15.604;
   1:L PR[91] R[100]mm/sec CNT100;
   1:  PR[91,1] = PR[90,1] + 30.084;
   1:  PR[91,2] = PR[90,2] + -12.608;
   1:L PR[91] R[100]mm/sec CNT100;
   1:  PR[91,1] = PR[90,1] + 30.423;
   1:  PR[91,2] = PR[90,2] + -12.167;
   1:L PR[91] R[100]mm/sec CNT100;
   1:  PR[91,1] = PR[90,1] + 32.268;
   1:  PR[91,2] = PR[90,2] + -9.295;
   1:L PR[91] R[100]mm/sec CNT100;
   1:  PR[91,1] = PR[90,1] + 32.623;
   1:  PR[91,2] = PR[90,2] + -8.669;
   1:L PR[91] R[100]mm/sec CNT100;
   1:  PR[91,1] = PR[90,1] + 32.912;
   1:  PR[91,2] = PR[90,2] + -7.935;
   1:L PR[91] R[100]mm/sec CNT100;
   1:  PR[91,1] = PR[90,1] + 33.983;
   1:  PR[91,2] = PR[90,2] + -5.021;
   1:L PR[91] R[100]mm/sec CNT100;
   1:  PR[91,1] = PR[90,1] + 34.130;
   1:  PR[91,2] = PR[90,2] + -4.376;
   1:L PR[91] R[100]mm/sec CNT100;
   1:  PR[91,1] = PR[90,1] + 34.197;
   1:  PR[91,2] = PR[90,2] + -3.439;
   1:L PR[91] R[100]mm/sec CNT100;
   1:  PR[91,1] = PR[90,1] + 34.550;
   1:  PR[91,2] = PR[90,2] + -0.371;
   1:L PR[91] R[100]mm/sec CNT100;
   1:  PR[91,1] = PR[90,1] + 34.492;
   1:  PR[91,2] = PR[90,2] + 0.443;
   1:L PR[91] R[100]mm/sec CNT100;
   1:  PR[91,1] = PR[90,1] + 34.142;
   1:  PR[91,2] = PR[90,2] + 3.477;
   1:L PR[91] R[100]mm/sec CNT100;
   1:  PR[91,1] = PR[90,1] + 33.990;
   1:  PR[91,2] = PR[90,2] + 4.146;
   1:L PR[91] R[100]mm/sec CNT100;
   1:  PR[91,1] = PR[90,1] + 33.678;
   1:  PR[91,2] = PR[90,2] + 4.936;
   1:L PR[91] R[100]mm/sec CNT100;
   1:  PR[91,1] = PR[90,1] + 32.609;
   1:  PR[91,2] = PR[90,2] + 7.846;
   1:L PR[91] R[100]mm/sec CNT100;
   1:  PR[91,1] = PR[90,1] + 32.268;
   1:  PR[91,2] = PR[90,2] + 8.448;
   1:L PR[91] R[100]mm/sec CNT100;
   1:  PR[91,1] = PR[90,1] + 30.423;
   1:  PR[91,2] = PR[90,2] + 11.319;
   1:L PR[91] R[100]mm/sec CNT100;
   1:  PR[91,1] = PR[90,1] + 30.084;
   1:  PR[91,2] = PR[90,2] + 11.760;
   1:L PR[91] R[100]mm/sec CNT100;
   1:  PR[91,1] = PR[90,1] + 27.029;
   1:  PR[91,2] = PR[90,2] + 14.757;
   1:L PR[91] R[100]mm/sec CNT100;
   1:  PR[91,1] = PR[90,1] + 26.758;
   1:  PR[91,2] = PR[90,2] + 14.956;
   1:L PR[91] R[100]mm/sec CNT100;
   1:  PR[91,1] = PR[90,1] + 23.223;
   1:  PR[91,2] = PR[90,2] + 17.155;
   1:L PR[91] R[100]mm/sec CNT100;
   1:  PR[91,1] = PR[90,1] + 23.067;
   1:  PR[91,2] = PR[90,2] + 17.240;
   1:L PR[91] R[100]mm/sec CNT100;
   1:  PR[91,1] = PR[90,1] + 22.898;
   1:  PR[91,2] = PR[90,2] + 17.304;
   1:L PR[91] R[100]mm/sec CNT100;
   1:  PR[91,1] = PR[90,1] + 18.679;
   1:  PR[91,2] = PR[90,2] + 18.817;
   1:L PR[91] R[100]mm/sec CNT100;
   1:  PR[91,1] = PR[90,1] + 16.062;
   1:  PR[91,2] = PR[90,2] + 19.165;
   1:L PR[91] R[100]mm/sec CNT100;
   1:  PR[91,1] = PR[90,1] + 14.021;
   1:  PR[91,2] = PR[90,2] + 19.460;
   1:L PR[91] R[100]mm/sec CNT100;
   1:  PR[91,1] = PR[90,1] + 9.353;
   1:  PR[91,2] = PR[90,2] + 19.141;
   1:L PR[91] R[100]mm/sec CNT100;
   1:  PR[91,1] = PR[90,1] + 8.974;
   1:  PR[91,2] = PR[90,2] + 19.042;
   1:L PR[91] R[100]mm/sec CNT100;
   1:  PR[91,1] = PR[90,1] + 4.892;
   1:  PR[91,2] = PR[90,2] + 17.848;
   1:L PR[91] R[100]mm/sec CNT100;
   1:  PR[91,1] = PR[90,1] + 3.243;
   1:  PR[91,2] = PR[90,2] + 17.014;
   1:L PR[91] R[100]mm/sec CNT100;
   1:  PR[91,1] = PR[90,1] + 1.901;
   1:  PR[91,2] = PR[90,2] + 16.280;
   1:L PR[91] R[100]mm/sec CNT100;
   1:  PR[91,1] = PR[90,1] + 1.474;
   1:  PR[91,2] = PR[90,2] + 15.975;
   1:L PR[91] R[100]mm/sec CNT100;
   1:  PR[91,1] = PR[90,1] + 0.765;
   1:  PR[91,2] = PR[90,2] + 15.867;
   1:L PR[91] R[100]mm/sec CNT100;
   1:  PR[91,1] = PR[90,1] + -0.280;
   1:  PR[91,2] = PR[90,2] + 15.503;
   1:L PR[91] R[100]mm/sec CNT100;
   1:  PR[91] = PR[90];
   1:  PR[91,1] = PR[90,1] + -2.025;
   1:  PR[91,2] = PR[90,2] + 16.594;
   1:  PR[91,3] = PR[90,3] + 40.495;
   1:L PR[91] R[100]mm/sec CNT100;
   1:  PR[91,1] = PR[90,1] + -4.725;
   1:  PR[91,2] = PR[90,2] + 17.979;
   1:L PR[91] R[100]mm/sec CNT100;
   1:  PR[91,1] = PR[90,1] + -4.857;
   1:  PR[91,2] = PR[90,2] + 18.039;
   1:L PR[91] R[100]mm/sec CNT100;
   1:  PR[91,1] = PR[90,1] + -8.429;
   1:  PR[91,2] = PR[90,2] + 19.084;
   1:L PR[91] R[100]mm/sec CNT100;
   1:  PR[91,1] = PR[90,1] + -9.399;
   1:  PR[91,2] = PR[90,2] + 19.338;
   1:L PR[91] R[100]mm/sec CNT100;
   1:  PR[91,1] = PR[90,1] + -13.509;
   1:  PR[91,2] = PR[90,2] + 19.622;
   1:L PR[91] R[100]mm/sec CNT100;
   1:  PR[91,1] = PR[90,1] + -14.054;
   1:  PR[91,2] = PR[90,2] + 19.644;
   1:L PR[91] R[100]mm/sec CNT100;
   1:  PR[91,1] = PR[90,1] + -18.704;
   1:  PR[91,2] = PR[90,2] + 18.964;
   1:L PR[91] R[100]mm/sec CNT100;
   1:  PR[91,1] = PR[90,1] + -23.069;
   1:  PR[91,2] = PR[90,2] + 17.352;
   1:L PR[91] R[100]mm/sec CNT100;
   1:  PR[91,1] = PR[90,1] + -26.990;
   1:  PR[91,2] = PR[90,2] + 14.912;
   1:L PR[91] R[100]mm/sec CNT100;
   1:  PR[91,1] = PR[90,1] + -30.212;
   1:  PR[91,2] = PR[90,2] + 11.754;
   1:L PR[91] R[100]mm/sec CNT100;
   1:  PR[91,1] = PR[90,1] + -30.325;
   1:  PR[91,2] = PR[90,2] + 11.607;
   1:L PR[91] R[100]mm/sec CNT100;
   1:  PR[91,1] = PR[90,1] + -32.487;
   1:  PR[91,2] = PR[90,2] + 8.236;
   1:L PR[91] R[100]mm/sec CNT100;
   1:  PR[91,1] = PR[90,1] + -32.661;
   1:  PR[91,2] = PR[90,2] + 7.928;
   1:L PR[91] R[100]mm/sec CNT100;
   1:  PR[91,1] = PR[90,1] + -32.817;
   1:  PR[91,2] = PR[90,2] + 7.527;
   1:L PR[91] R[100]mm/sec CNT100;
   1:  PR[91,1] = PR[90,1] + -34.093;
   1:  PR[91,2] = PR[90,2] + 4.041;
   1:L PR[91] R[100]mm/sec CNT100;
   1:  PR[91,1] = PR[90,1] + -34.163;
   1:  PR[91,2] = PR[90,2] + 3.730;
   1:L PR[91] R[100]mm/sec CNT100;
   1:  PR[91,1] = PR[90,1] + -34.201;
   1:  PR[91,2] = PR[90,2] + 3.180;
   1:L PR[91] R[100]mm/sec CNT100;
   1:  PR[91,1] = PR[90,1] + -34.623;
   1:  PR[91,2] = PR[90,2] + -0.479;
   1:L PR[91] R[100]mm/sec CNT100;
   1:  PR[91,1] = PR[90,1] + -34.593;
   1:  PR[91,2] = PR[90,2] + -0.908;
   1:L PR[91] R[100]mm/sec CNT100;
   1:  PR[91,1] = PR[90,1] + -34.175;
   1:  PR[91,2] = PR[90,2] + -4.523;
   1:L PR[91] R[100]mm/sec CNT100;
   1:  PR[91,1] = PR[90,1] + -34.098;
   1:  PR[91,2] = PR[90,2] + -4.864;
   1:L PR[91] R[100]mm/sec CNT100;
   1:  PR[91,1] = PR[90,1] + -33.913;
   1:  PR[91,2] = PR[90,2] + -5.339;
   1:L PR[91] R[100]mm/sec CNT100;
   1:  PR[91,1] = PR[90,1] + -32.649;
   1:  PR[91,2] = PR[90,2] + -8.796;
   1:L PR[91] R[100]mm/sec CNT100;
   1:  PR[91,1] = PR[90,1] + -32.487;
   1:  PR[91,2] = PR[90,2] + -9.084;
   1:L PR[91] R[100]mm/sec CNT100;
   1:  PR[91,1] = PR[90,1] + -30.325;
   1:  PR[91,2] = PR[90,2] + -12.455;
   1:L PR[91] R[100]mm/sec CNT100;
   1:  PR[91,1] = PR[90,1] + -30.212;
   1:  PR[91,2] = PR[90,2] + -12.602;
   1:L PR[91] R[100]mm/sec CNT100;
   1:  PR[91,1] = PR[90,1] + -26.990;
   1:  PR[91,2] = PR[90,2] + -15.759;
   1:L PR[91] R[100]mm/sec CNT100;
   1:  PR[91,1] = PR[90,1] + -23.069;
   1:  PR[91,2] = PR[90,2] + -18.199;
   1:L PR[91] R[100]mm/sec CNT100;
   1:  PR[91,1] = PR[90,1] + -18.703;
   1:  PR[91,2] = PR[90,2] + -19.811;
   1:L PR[91] R[100]mm/sec CNT100;
   1:  PR[91,1] = PR[90,1] + -14.054;
   1:  PR[91,2] = PR[90,2] + -20.491;
   1:L PR[91] R[100]mm/sec CNT100;
   1:  PR[91,1] = PR[90,1] + -13.509;
   1:  PR[91,2] = PR[90,2] + -20.469;
   1:L PR[91] R[100]mm/sec CNT100;
   1:  PR[91,1] = PR[90,1] + -9.399;
   1:  PR[91,2] = PR[90,2] + -20.185;
   1:L PR[91] R[100]mm/sec CNT100;
   1:  PR[91,1] = PR[90,1] + -8.428;
   1:  PR[91,2] = PR[90,2] + -19.931;
   1:L PR[91] R[100]mm/sec CNT100;
   1:  PR[91,1] = PR[90,1] + -4.857;
   1:  PR[91,2] = PR[90,2] + -18.886;
   1:L PR[91] R[100]mm/sec CNT100;
   1:  PR[91,1] = PR[90,1] + -4.706;
   1:  PR[91,2] = PR[90,2] + -18.817;
   1:L PR[91] R[100]mm/sec CNT100;
   1:  PR[91,1] = PR[90,1] + -2.024;
   1:  PR[91,2] = PR[90,2] + -17.439;
   1:L PR[91] R[100]mm/sec CNT100;
   1:  PR[91,1] = PR[90,1] + -0.255;
   1:  PR[91,2] = PR[90,2] + -16.814;
   1:L PR[91] R[100]mm/sec CNT100;
   1:  PR[91,1] = PR[90,1] + 1.534;
   1:  PR[91,2] = PR[90,2] + -17.437;
   1:L PR[91] R[100]mm/sec CNT100;
   1:  PR[91,1] = PR[90,1] + 4.221;
   1:  PR[91,2] = PR[90,2] + -18.815;
   1:L PR[91] R[100]mm/sec CNT100;
   1:  PR[91,1] = PR[90,1] + 4.374;
   1:  PR[91,2] = PR[90,2] + -18.885;
   1:L PR[91] R[100]mm/sec CNT100;
   1:  PR[91,1] = PR[90,1] + 7.945;
   1:  PR[91,2] = PR[90,2] + -19.929;
   1:L PR[91] R[100]mm/sec CNT100;
   1:  PR[91,1] = PR[90,1] + 8.916;
   1:  PR[91,2] = PR[90,2] + -20.184;
   1:L PR[91] R[100]mm/sec CNT100;
   1:  PR[91,1] = PR[90,1] + 13.027;
   1:  PR[91,2] = PR[90,2] + -20.469;
   1:L PR[91] R[100]mm/sec CNT100;
   1:  PR[91,1] = PR[90,1] + 13.571;
   1:  PR[91,2] = PR[90,2] + -20.492;
   1:L PR[91] R[100]mm/sec CNT100;
   1:  PR[91,1] = PR[90,1] + 18.221;
   1:  PR[91,2] = PR[90,2] + -19.811;
   1:L PR[91] R[100]mm/sec CNT100;
   1:  PR[91,1] = PR[90,1] + 22.588;
   1:  PR[91,2] = PR[90,2] + -18.200;
   1:L PR[91] R[100]mm/sec CNT100;
   1:  PR[91,1] = PR[90,1] + 26.506;
   1:  PR[91,2] = PR[90,2] + -15.765;
   1:L PR[91] R[100]mm/sec CNT100;
   1:  PR[91,1] = PR[90,1] + 29.724;
   1:  PR[91,2] = PR[90,2] + -12.604;
   1:L PR[91] R[100]mm/sec CNT100;
   1:  PR[91,1] = PR[90,1] + 29.841;
   1:  PR[91,2] = PR[90,2] + -12.452;
   1:L PR[91] R[100]mm/sec CNT100;
   1:  PR[91,1] = PR[90,1] + 32.005;
   1:  PR[91,2] = PR[90,2] + -9.084;
   1:L PR[91] R[100]mm/sec CNT100;
   1:  PR[91,1] = PR[90,1] + 32.182;
   1:  PR[91,2] = PR[90,2] + -8.772;
   1:L PR[91] R[100]mm/sec CNT100;
   1:  PR[91,1] = PR[90,1] + 32.335;
   1:  PR[91,2] = PR[90,2] + -8.384;
   1:L PR[91] R[100]mm/sec CNT100;
   1:  PR[91,1] = PR[90,1] + 33.610;
   1:  PR[91,2] = PR[90,2] + -4.915;
   1:L PR[91] R[100]mm/sec CNT100;
   1:  PR[91,1] = PR[90,1] + 33.680;
   1:  PR[91,2] = PR[90,2] + -4.607;
   1:L PR[91] R[100]mm/sec CNT100;
   1:  PR[91,1] = PR[90,1] + 33.721;
   1:  PR[91,2] = PR[90,2] + -4.040;
   1:L PR[91] R[100]mm/sec CNT100;
   1:  PR[91,1] = PR[90,1] + 34.143;
   1:  PR[91,2] = PR[90,2] + -0.371;
   1:L PR[91] R[100]mm/sec CNT100;
   1:  PR[91,1] = PR[90,1] + 34.111;
   1:  PR[91,2] = PR[90,2] + 0.082;
   1:L PR[91] R[100]mm/sec CNT100;
   1:  PR[91,1] = PR[90,1] + 33.692;
   1:  PR[91,2] = PR[90,2] + 3.709;
   1:L PR[91] R[100]mm/sec CNT100;
   1:  PR[91,1] = PR[90,1] + 33.617;
   1:  PR[91,2] = PR[90,2] + 4.040;
   1:L PR[91] R[100]mm/sec CNT100;
   1:  PR[91,1] = PR[90,1] + 33.432;
   1:  PR[91,2] = PR[90,2] + 4.507;
   1:L PR[91] R[100]mm/sec CNT100;
   1:  PR[91,1] = PR[90,1] + 32.168;
   1:  PR[91,2] = PR[90,2] + 7.949;
   1:L PR[91] R[100]mm/sec CNT100;
   1:  PR[91,1] = PR[90,1] + 32.005;
   1:  PR[91,2] = PR[90,2] + 8.237;
   1:L PR[91] R[100]mm/sec CNT100;
   1:  PR[91,1] = PR[90,1] + 29.841;
   1:  PR[91,2] = PR[90,2] + 11.605;
   1:L PR[91] R[100]mm/sec CNT100;
   1:  PR[91,1] = PR[90,1] + 29.724;
   1:  PR[91,2] = PR[90,2] + 11.757;
   1:L PR[91] R[100]mm/sec CNT100;
   1:  PR[91,1] = PR[90,1] + 26.506;
   1:  PR[91,2] = PR[90,2] + 14.918;
   1:L PR[91] R[100]mm/sec CNT100;
   1:  PR[91,1] = PR[90,1] + 22.588;
   1:  PR[91,2] = PR[90,2] + 17.352;
   1:L PR[91] R[100]mm/sec CNT100;
   1:  PR[91,1] = PR[90,1] + 18.221;
   1:  PR[91,2] = PR[90,2] + 18.964;
   1:L PR[91] R[100]mm/sec CNT100;
   1:  PR[91,1] = PR[90,1] + 13.571;
   1:  PR[91,2] = PR[90,2] + 19.645;
   1:L PR[91] R[100]mm/sec CNT100;
   1:  PR[91,1] = PR[90,1] + 13.027;
   1:  PR[91,2] = PR[90,2] + 19.622;
   1:L PR[91] R[100]mm/sec CNT100;
   1:  PR[91,1] = PR[90,1] + 8.917;
   1:  PR[91,2] = PR[90,2] + 19.337;
   1:L PR[91] R[100]mm/sec CNT100;
   1:  PR[91,1] = PR[90,1] + 7.946;
   1:  PR[91,2] = PR[90,2] + 19.082;
   1:L PR[91] R[100]mm/sec CNT100;
   1:  PR[91,1] = PR[90,1] + 4.374;
   1:  PR[91,2] = PR[90,2] + 18.037;
   1:L PR[91] R[100]mm/sec CNT100;
   1:  PR[91,1] = PR[90,1] + 4.240;
   1:  PR[91,2] = PR[90,2] + 17.976;
   1:L PR[91] R[100]mm/sec CNT100;
   1:  PR[91,1] = PR[90,1] + 1.530;
   1:  PR[91,2] = PR[90,2] + 16.589;
   1:L PR[91] R[100]mm/sec CNT100;
   1:  PR[91,1] = PR[90,1] + -0.258;
   1:  PR[91,2] = PR[90,2] + 15.966;
   1:L PR[91] R[100]mm/sec CNT100;
   1:  PR[91] = PR[90];
   1:  PR[91,1] = PR[90,1] + -1.438;
   1:  PR[91,2] = PR[90,2] + 16.869;
   1:  PR[91,3] = PR[90,3] + 41.795;
   1:L PR[91] R[100]mm/sec CNT100;
   1:  PR[91,1] = PR[90,1] + -1.781;
   1:  PR[91,2] = PR[90,2] + 16.921;
   1:L PR[91] R[100]mm/sec CNT100;
   1:  PR[91,1] = PR[90,1] + -4.131;
   1:  PR[91,2] = PR[90,2] + 18.127;
   1:L PR[91] R[100]mm/sec CNT100;
   1:  PR[91,1] = PR[90,1] + -4.386;
   1:  PR[91,2] = PR[90,2] + 18.243;
   1:L PR[91] R[100]mm/sec CNT100;
   1:  PR[91,1] = PR[90,1] + -7.401;
   1:  PR[91,2] = PR[90,2] + 19.124;
   1:L PR[91] R[100]mm/sec CNT100;
   1:  PR[91,1] = PR[90,1] + -8.961;
   1:  PR[91,2] = PR[90,2] + 19.534;
   1:L PR[91] R[100]mm/sec CNT100;
   1:  PR[91,1] = PR[90,1] + -12.491;
   1:  PR[91,2] = PR[90,2] + 19.777;
   1:L PR[91] R[100]mm/sec CNT100;
   1:  PR[91,1] = PR[90,1] + -13.641;
   1:  PR[91,2] = PR[90,2] + 19.824;
   1:L PR[91] R[100]mm/sec CNT100;
   1:  PR[91,1] = PR[90,1] + -17.559;
   1:  PR[91,2] = PR[90,2] + 19.259;
   1:L PR[91] R[100]mm/sec CNT100;
   1:  PR[91,1] = PR[90,1] + -18.279;
   1:  PR[91,2] = PR[90,2] + 19.136;
   1:L PR[91] R[100]mm/sec CNT100;
   1:  PR[91,1] = PR[90,1] + -22.359;
   1:  PR[91,2] = PR[90,2] + 17.621;
   1:L PR[91] R[100]mm/sec CNT100;
   1:  PR[91,1] = PR[90,1] + -22.645;
   1:  PR[91,2] = PR[90,2] + 17.507;
   1:L PR[91] R[100]mm/sec CNT100;
   1:  PR[91,1] = PR[90,1] + -26.550;
   1:  PR[91,2] = PR[90,2] + 15.015;
   1:L PR[91] R[100]mm/sec CNT100;
   1:  PR[91,1] = PR[90,1] + -28.204;
   1:  PR[91,2] = PR[90,2] + 13.368;
   1:L PR[91] R[100]mm/sec CNT100;
   1:  PR[91,1] = PR[90,1] + -29.776;
   1:  PR[91,2] = PR[90,2] + 11.827;
   1:L PR[91] R[100]mm/sec CNT100;
   1:  PR[91,1] = PR[90,1] + -32.210;
   1:  PR[91,2] = PR[90,2] + 8.046;
   1:L PR[91] R[100]mm/sec CNT100;
   1:  PR[91,1] = PR[90,1] + -33.712;
   1:  PR[91,2] = PR[90,2] + 3.956;
   1:L PR[91] R[100]mm/sec CNT100;
   1:  PR[91,1] = PR[90,1] + -33.725;
   1:  PR[91,2] = PR[90,2] + 3.779;
   1:L PR[91] R[100]mm/sec CNT100;
   1:  PR[91,1] = PR[90,1] + -34.216;
   1:  PR[91,2] = PR[90,2] + -0.479;
   1:L PR[91] R[100]mm/sec CNT100;
   1:  PR[91,1] = PR[90,1] + -34.210;
   1:  PR[91,2] = PR[90,2] + -0.558;
   1:L PR[91] R[100]mm/sec CNT100;
   1:  PR[91,1] = PR[90,1] + -33.723;
   1:  PR[91,2] = PR[90,2] + -4.764;
   1:L PR[91] R[100]mm/sec CNT100;
   1:  PR[91,1] = PR[90,1] + -33.666;
   1:  PR[91,2] = PR[90,2] + -4.912;
   1:L PR[91] R[100]mm/sec CNT100;
   1:  PR[91,1] = PR[90,1] + -32.209;
   1:  PR[91,2] = PR[90,2] + -8.895;
   1:L PR[91] R[100]mm/sec CNT100;
   1:  PR[91,1] = PR[90,1] + -29.776;
   1:  PR[91,2] = PR[90,2] + -12.674;
   1:L PR[91] R[100]mm/sec CNT100;
   1:  PR[91,1] = PR[90,1] + -28.204;
   1:  PR[91,2] = PR[90,2] + -14.215;
   1:L PR[91] R[100]mm/sec CNT100;
   1:  PR[91,1] = PR[90,1] + -26.550;
   1:  PR[91,2] = PR[90,2] + -15.863;
   1:L PR[91] R[100]mm/sec CNT100;
   1:  PR[91,1] = PR[90,1] + -22.645;
   1:  PR[91,2] = PR[90,2] + -18.355;
   1:L PR[91] R[100]mm/sec CNT100;
   1:  PR[91,1] = PR[90,1] + -22.359;
   1:  PR[91,2] = PR[90,2] + -18.469;
   1:L PR[91] R[100]mm/sec CNT100;
   1:  PR[91,1] = PR[90,1] + -18.278;
   1:  PR[91,2] = PR[90,2] + -19.983;
   1:L PR[91] R[100]mm/sec CNT100;
   1:  PR[91,1] = PR[90,1] + -17.558;
   1:  PR[91,2] = PR[90,2] + -20.106;
   1:L PR[91] R[100]mm/sec CNT100;
   1:  PR[91,1] = PR[90,1] + -13.641;
   1:  PR[91,2] = PR[90,2] + -20.672;
   1:L PR[91] R[100]mm/sec CNT100;
   1:  PR[91,1] = PR[90,1] + -12.490;
   1:  PR[91,2] = PR[90,2] + -20.624;
   1:L PR[91] R[100]mm/sec CNT100;
   1:  PR[91,1] = PR[90,1] + -8.960;
   1:  PR[91,2] = PR[90,2] + -20.381;
   1:L PR[91] R[100]mm/sec CNT100;
   1:  PR[91,1] = PR[90,1] + -7.399;
   1:  PR[91,2] = PR[90,2] + -19.971;
   1:L PR[91] R[100]mm/sec CNT100;
   1:  PR[91,1] = PR[90,1] + -4.385;
   1:  PR[91,2] = PR[90,2] + -19.090;
   1:L PR[91] R[100]mm/sec CNT100;
   1:  PR[91,1] = PR[90,1] + -4.105;
   1:  PR[91,2] = PR[90,2] + -18.962;
   1:L PR[91] R[100]mm/sec CNT100;
   1:  PR[91,1] = PR[90,1] + -1.784;
   1:  PR[91,2] = PR[90,2] + -17.769;
   1:L PR[91] R[100]mm/sec CNT100;
   1:  PR[91,1] = PR[90,1] + -1.434;
   1:  PR[91,2] = PR[90,2] + -17.715;
   1:L PR[91] R[100]mm/sec CNT100;
   1:  PR[91,1] = PR[90,1] + -0.229;
   1:  PR[91,2] = PR[90,2] + -17.287;
   1:L PR[91] R[100]mm/sec CNT100;
   1:  PR[91,1] = PR[90,1] + 1.487;
   1:  PR[91,2] = PR[90,2] + -17.866;
   1:L PR[91] R[100]mm/sec CNT100;
   1:  PR[91,1] = PR[90,1] + 3.621;
   1:  PR[91,2] = PR[90,2] + -18.960;
   1:L PR[91] R[100]mm/sec CNT100;
   1:  PR[91,1] = PR[90,1] + 3.903;
   1:  PR[91,2] = PR[90,2] + -19.088;
   1:L PR[91] R[100]mm/sec CNT100;
   1:  PR[91,1] = PR[90,1] + 6.917;
   1:  PR[91,2] = PR[90,2] + -19.970;
   1:L PR[91] R[100]mm/sec CNT100;
   1:  PR[91,1] = PR[90,1] + 8.478;
   1:  PR[91,2] = PR[90,2] + -20.380;
   1:L PR[91] R[100]mm/sec CNT100;
   1:  PR[91,1] = PR[90,1] + 12.008;
   1:  PR[91,2] = PR[90,2] + -20.625;
   1:L PR[91] R[100]mm/sec CNT100;
   1:  PR[91,1] = PR[90,1] + 13.158;
   1:  PR[91,2] = PR[90,2] + -20.672;
   1:L PR[91] R[100]mm/sec CNT100;
   1:  PR[91,1] = PR[90,1] + 17.075;
   1:  PR[91,2] = PR[90,2] + -20.106;
   1:L PR[91] R[100]mm/sec CNT100;
   1:  PR[91,1] = PR[90,1] + 17.796;
   1:  PR[91,2] = PR[90,2] + -19.983;
   1:L PR[91] R[100]mm/sec CNT100;
   1:  PR[91,1] = PR[90,1] + 21.878;
   1:  PR[91,2] = PR[90,2] + -18.469;
   1:L PR[91] R[100]mm/sec CNT100;
   1:  PR[91,1] = PR[90,1] + 22.165;
   1:  PR[91,2] = PR[90,2] + -18.355;
   1:L PR[91] R[100]mm/sec CNT100;
   1:  PR[91,1] = PR[90,1] + 26.055;
   1:  PR[91,2] = PR[90,2] + -15.880;
   1:L PR[91] R[100]mm/sec CNT100;
   1:  PR[91,1] = PR[90,1] + 27.721;
   1:  PR[91,2] = PR[90,2] + -14.216;
   1:L PR[91] R[100]mm/sec CNT100;
   1:  PR[91,1] = PR[90,1] + 29.318;
   1:  PR[91,2] = PR[90,2] + -12.647;
   1:L PR[91] R[100]mm/sec CNT100;
   1:  PR[91,1] = PR[90,1] + 31.731;
   1:  PR[91,2] = PR[90,2] + -8.891;
   1:L PR[91] R[100]mm/sec CNT100;
   1:  PR[91,1] = PR[90,1] + 33.232;
   1:  PR[91,2] = PR[90,2] + -4.824;
   1:L PR[91] R[100]mm/sec CNT100;
   1:  PR[91,1] = PR[90,1] + 33.245;
   1:  PR[91,2] = PR[90,2] + -4.641;
   1:L PR[91] R[100]mm/sec CNT100;
   1:  PR[91,1] = PR[90,1] + 33.736;
   1:  PR[91,2] = PR[90,2] + -0.371;
   1:L PR[91] R[100]mm/sec CNT100;
   1:  PR[91,1] = PR[90,1] + 33.729;
   1:  PR[91,2] = PR[90,2] + -0.279;
   1:L PR[91] R[100]mm/sec CNT100;
   1:  PR[91,1] = PR[90,1] + 33.242;
   1:  PR[91,2] = PR[90,2] + 3.940;
   1:L PR[91] R[100]mm/sec CNT100;
   1:  PR[91,1] = PR[90,1] + 33.238;
   1:  PR[91,2] = PR[90,2] + 3.961;
   1:L PR[91] R[100]mm/sec CNT100;
   1:  PR[91,1] = PR[90,1] + 31.731;
   1:  PR[91,2] = PR[90,2] + 8.043;
   1:L PR[91] R[100]mm/sec CNT100;
   1:  PR[91,1] = PR[90,1] + 29.293;
   1:  PR[91,2] = PR[90,2] + 11.823;
   1:L PR[91] R[100]mm/sec CNT100;
   1:  PR[91,1] = PR[90,1] + 27.721;
   1:  PR[91,2] = PR[90,2] + 13.369;
   1:L PR[91] R[100]mm/sec CNT100;
   1:  PR[91,1] = PR[90,1] + 26.056;
   1:  PR[91,2] = PR[90,2] + 15.032;
   1:L PR[91] R[100]mm/sec CNT100;
   1:  PR[91,1] = PR[90,1] + 22.165;
   1:  PR[91,2] = PR[90,2] + 17.508;
   1:L PR[91] R[100]mm/sec CNT100;
   1:  PR[91,1] = PR[90,1] + 21.878;
   1:  PR[91,2] = PR[90,2] + 17.622;
   1:L PR[91] R[100]mm/sec CNT100;
   1:  PR[91,1] = PR[90,1] + 17.796;
   1:  PR[91,2] = PR[90,2] + 19.135;
   1:L PR[91] R[100]mm/sec CNT100;
   1:  PR[91,1] = PR[90,1] + 17.075;
   1:  PR[91,2] = PR[90,2] + 19.259;
   1:L PR[91] R[100]mm/sec CNT100;
   1:  PR[91,1] = PR[90,1] + 13.158;
   1:  PR[91,2] = PR[90,2] + 19.825;
   1:L PR[91] R[100]mm/sec CNT100;
   1:  PR[91,1] = PR[90,1] + 12.008;
   1:  PR[91,2] = PR[90,2] + 19.777;
   1:L PR[91] R[100]mm/sec CNT100;
   1:  PR[91,1] = PR[90,1] + 8.479;
   1:  PR[91,2] = PR[90,2] + 19.533;
   1:L PR[91] R[100]mm/sec CNT100;
   1:  PR[91,1] = PR[90,1] + 6.919;
   1:  PR[91,2] = PR[90,2] + 19.123;
   1:L PR[91] R[100]mm/sec CNT100;
   1:  PR[91,1] = PR[90,1] + 3.903;
   1:  PR[91,2] = PR[90,2] + 18.241;
   1:L PR[91] R[100]mm/sec CNT100;
   1:  PR[91,1] = PR[90,1] + 3.647;
   1:  PR[91,2] = PR[90,2] + 18.125;
   1:L PR[91] R[100]mm/sec CNT100;
   1:  PR[91,1] = PR[90,1] + 1.486;
   1:  PR[91,2] = PR[90,2] + 17.018;
   1:L PR[91] R[100]mm/sec CNT100;
   1:  PR[91,1] = PR[90,1] + -0.230;
   1:  PR[91,2] = PR[90,2] + 16.440;
   1:L PR[91] R[100]mm/sec CNT100;
   1:  PR[91] = PR[90];
   1:  PR[91,1] = PR[90,1] + -1.219;
   1:  PR[91,2] = PR[90,2] + 17.275;
   1:  PR[91,3] = PR[90,3] + 43.095;
   1:L PR[91] R[100]mm/sec CNT100;
   1:  PR[91,1] = PR[90,1] + -1.745;
   1:  PR[91,2] = PR[90,2] + 17.355;
   1:L PR[91] R[100]mm/sec CNT100;
   1:  PR[91,1] = PR[90,1] + -3.537;
   1:  PR[91,2] = PR[90,2] + 18.275;
   1:L PR[91] R[100]mm/sec CNT100;
   1:  PR[91,1] = PR[90,1] + -3.914;
   1:  PR[91,2] = PR[90,2] + 18.446;
   1:L PR[91] R[100]mm/sec CNT100;
   1:  PR[91,1] = PR[90,1] + -6.372;
   1:  PR[91,2] = PR[90,2] + 19.165;
   1:L PR[91] R[100]mm/sec CNT100;
   1:  PR[91,1] = PR[90,1] + -8.522;
   1:  PR[91,2] = PR[90,2] + 19.729;
   1:L PR[91] R[100]mm/sec CNT100;
   1:  PR[91,1] = PR[90,1] + -11.472;
   1:  PR[91,2] = PR[90,2] + 19.932;
   1:L PR[91] R[100]mm/sec CNT100;
   1:  PR[91,1] = PR[90,1] + -13.226;
   1:  PR[91,2] = PR[90,2] + 20.005;
   1:L PR[91] R[100]mm/sec CNT100;
   1:  PR[91,1] = PR[90,1] + -16.552;
   1:  PR[91,2] = PR[90,2] + 19.524;
   1:L PR[91] R[100]mm/sec CNT100;
   1:  PR[91,1] = PR[90,1] + -17.883;
   1:  PR[91,2] = PR[90,2] + 19.297;
   1:L PR[91] R[100]mm/sec CNT100;
   1:  PR[91,1] = PR[90,1] + -21.392;
   1:  PR[91,2] = PR[90,2] + 17.995;
   1:L PR[91] R[100]mm/sec CNT100;
   1:  PR[91,1] = PR[90,1] + -22.266;
   1:  PR[91,2] = PR[90,2] + 17.646;
   1:L PR[91] R[100]mm/sec CNT100;
   1:  PR[91,1] = PR[90,1] + -25.707;
   1:  PR[91,2] = PR[90,2] + 15.454;
   1:L PR[91] R[100]mm/sec CNT100;
   1:  PR[91,1] = PR[90,1] + -26.164;
   1:  PR[91,2] = PR[90,2] + 15.148;
   1:L PR[91] R[100]mm/sec CNT100;
   1:  PR[91,1] = PR[90,1] + -29.245;
   1:  PR[91,2] = PR[90,2] + 12.079;
   1:L PR[91] R[100]mm/sec CNT100;
   1:  PR[91,1] = PR[90,1] + -29.390;
   1:  PR[91,2] = PR[90,2] + 11.928;
   1:L PR[91] R[100]mm/sec CNT100;
   1:  PR[91,1] = PR[90,1] + -31.815;
   1:  PR[91,2] = PR[90,2] + 8.091;
   1:L PR[91] R[100]mm/sec CNT100;
   1:  PR[91,1] = PR[90,1] + -33.300;
   1:  PR[91,2] = PR[90,2] + 3.984;
   1:L PR[91] R[100]mm/sec CNT100;
   1:  PR[91,1] = PR[90,1] + -33.803;
   1:  PR[91,2] = PR[90,2] + -0.424;
   1:L PR[91] R[100]mm/sec CNT100;
   1:  PR[91,1] = PR[90,1] + -33.300;
   1:  PR[91,2] = PR[90,2] + -4.831;
   1:L PR[91] R[100]mm/sec CNT100;
   1:  PR[91,1] = PR[90,1] + -31.815;
   1:  PR[91,2] = PR[90,2] + -8.938;
   1:L PR[91] R[100]mm/sec CNT100;
   1:  PR[91,1] = PR[90,1] + -29.402;
   1:  PR[91,2] = PR[90,2] + -12.757;
   1:L PR[91] R[100]mm/sec CNT100;
   1:  PR[91,1] = PR[90,1] + -26.161;
   1:  PR[91,2] = PR[90,2] + -15.997;
   1:L PR[91] R[100]mm/sec CNT100;
   1:  PR[91,1] = PR[90,1] + -25.707;
   1:  PR[91,2] = PR[90,2] + -16.301;
   1:L PR[91] R[100]mm/sec CNT100;
   1:  PR[91,1] = PR[90,1] + -22.265;
   1:  PR[91,2] = PR[90,2] + -18.494;
   1:L PR[91] R[100]mm/sec CNT100;
   1:  PR[91,1] = PR[90,1] + -21.392;
   1:  PR[91,2] = PR[90,2] + -18.842;
   1:L PR[91] R[100]mm/sec CNT100;
   1:  PR[91,1] = PR[90,1] + -17.882;
   1:  PR[91,2] = PR[90,2] + -20.144;
   1:L PR[91] R[100]mm/sec CNT100;
   1:  PR[91,1] = PR[90,1] + -16.551;
   1:  PR[91,2] = PR[90,2] + -20.372;
   1:L PR[91] R[100]mm/sec CNT100;
   1:  PR[91,1] = PR[90,1] + -13.225;
   1:  PR[91,2] = PR[90,2] + -20.852;
   1:L PR[91] R[100]mm/sec CNT100;
   1:  PR[91,1] = PR[90,1] + -11.471;
   1:  PR[91,2] = PR[90,2] + -20.780;
   1:L PR[91] R[100]mm/sec CNT100;
   1:  PR[91,1] = PR[90,1] + -8.522;
   1:  PR[91,2] = PR[90,2] + -20.576;
   1:L PR[91] R[100]mm/sec CNT100;
   1:  PR[91,1] = PR[90,1] + -6.370;
   1:  PR[91,2] = PR[90,2] + -20.011;
   1:L PR[91] R[100]mm/sec CNT100;
   1:  PR[91,1] = PR[90,1] + -3.914;
   1:  PR[91,2] = PR[90,2] + -19.293;
   1:L PR[91] R[100]mm/sec CNT100;
   1:  PR[91,1] = PR[90,1] + -3.504;
   1:  PR[91,2] = PR[90,2] + -19.106;
   1:L PR[91] R[100]mm/sec CNT100;
   1:  PR[91,1] = PR[90,1] + -1.748;
   1:  PR[91,2] = PR[90,2] + -18.204;
   1:L PR[91] R[100]mm/sec CNT100;
   1:  PR[91,1] = PR[90,1] + -1.216;
   1:  PR[91,2] = PR[90,2] + -18.122;
   1:L PR[91] R[100]mm/sec CNT100;
   1:  PR[91,1] = PR[90,1] + -0.175;
   1:  PR[91,2] = PR[90,2] + -17.752;
   1:L PR[91] R[100]mm/sec CNT100;
   1:  PR[91,1] = PR[90,1] + 1.011;
   1:  PR[91,2] = PR[90,2] + -18.165;
   1:L PR[91] R[100]mm/sec CNT100;
   1:  PR[91,1] = PR[90,1] + 1.382;
   1:  PR[91,2] = PR[90,2] + -18.265;
   1:L PR[91] R[100]mm/sec CNT100;
   1:  PR[91,1] = PR[90,1] + 3.021;
   1:  PR[91,2] = PR[90,2] + -19.104;
   1:L PR[91] R[100]mm/sec CNT100;
   1:  PR[91,1] = PR[90,1] + 3.432;
   1:  PR[91,2] = PR[90,2] + -19.292;
   1:L PR[91] R[100]mm/sec CNT100;
   1:  PR[91,1] = PR[90,1] + 5.889;
   1:  PR[91,2] = PR[90,2] + -20.011;
   1:L PR[91] R[100]mm/sec CNT100;
   1:  PR[91,1] = PR[90,1] + 8.040;
   1:  PR[91,2] = PR[90,2] + -20.575;
   1:L PR[91] R[100]mm/sec CNT100;
   1:  PR[91,1] = PR[90,1] + 10.990;
   1:  PR[91,2] = PR[90,2] + -20.780;
   1:L PR[91] R[100]mm/sec CNT100;
   1:  PR[91,1] = PR[90,1] + 12.743;
   1:  PR[91,2] = PR[90,2] + -20.852;
   1:L PR[91] R[100]mm/sec CNT100;
   1:  PR[91,1] = PR[90,1] + 16.069;
   1:  PR[91,2] = PR[90,2] + -20.372;
   1:L PR[91] R[100]mm/sec CNT100;
   1:  PR[91,1] = PR[90,1] + 17.401;
   1:  PR[91,2] = PR[90,2] + -20.144;
   1:L PR[91] R[100]mm/sec CNT100;
   1:  PR[91,1] = PR[90,1] + 20.911;
   1:  PR[91,2] = PR[90,2] + -18.843;
   1:L PR[91] R[100]mm/sec CNT100;
   1:  PR[91,1] = PR[90,1] + 21.785;
   1:  PR[91,2] = PR[90,2] + -18.494;
   1:L PR[91] R[100]mm/sec CNT100;
   1:  PR[91,1] = PR[90,1] + 25.226;
   1:  PR[91,2] = PR[90,2] + -16.305;
   1:L PR[91] R[100]mm/sec CNT100;
   1:  PR[91,1] = PR[90,1] + 25.679;
   1:  PR[91,2] = PR[90,2] + -16.002;
   1:L PR[91] R[100]mm/sec CNT100;
   1:  PR[91,1] = PR[90,1] + 28.921;
   1:  PR[91,2] = PR[90,2] + -12.752;
   1:L PR[91] R[100]mm/sec CNT100;
   1:  PR[91,1] = PR[90,1] + 31.336;
   1:  PR[91,2] = PR[90,2] + -8.935;
   1:L PR[91] R[100]mm/sec CNT100;
   1:  PR[91,1] = PR[90,1] + 32.820;
   1:  PR[91,2] = PR[90,2] + -4.849;
   1:L PR[91] R[100]mm/sec CNT100;
   1:  PR[91,1] = PR[90,1] + 33.323;
   1:  PR[91,2] = PR[90,2] + -0.424;
   1:L PR[91] R[100]mm/sec CNT100;
   1:  PR[91,1] = PR[90,1] + 32.820;
   1:  PR[91,2] = PR[90,2] + 4.001;
   1:L PR[91] R[100]mm/sec CNT100;
   1:  PR[91,1] = PR[90,1] + 31.336;
   1:  PR[91,2] = PR[90,2] + 8.088;
   1:L PR[91] R[100]mm/sec CNT100;
   1:  PR[91,1] = PR[90,1] + 28.921;
   1:  PR[91,2] = PR[90,2] + 11.905;
   1:L PR[91] R[100]mm/sec CNT100;
   1:  PR[91,1] = PR[90,1] + 25.679;
   1:  PR[91,2] = PR[90,2] + 15.155;
   1:L PR[91] R[100]mm/sec CNT100;
   1:  PR[91,1] = PR[90,1] + 25.226;
   1:  PR[91,2] = PR[90,2] + 15.458;
   1:L PR[91] R[100]mm/sec CNT100;
   1:  PR[91,1] = PR[90,1] + 21.785;
   1:  PR[91,2] = PR[90,2] + 17.647;
   1:L PR[91] R[100]mm/sec CNT100;
   1:  PR[91,1] = PR[90,1] + 20.911;
   1:  PR[91,2] = PR[90,2] + 17.995;
   1:L PR[91] R[100]mm/sec CNT100;
   1:  PR[91,1] = PR[90,1] + 17.401;
   1:  PR[91,2] = PR[90,2] + 19.297;
   1:L PR[91] R[100]mm/sec CNT100;
   1:  PR[91,1] = PR[90,1] + 16.069;
   1:  PR[91,2] = PR[90,2] + 19.524;
   1:L PR[91] R[100]mm/sec CNT100;
   1:  PR[91,1] = PR[90,1] + 12.743;
   1:  PR[91,2] = PR[90,2] + 20.005;
   1:L PR[91] R[100]mm/sec CNT100;
   1:  PR[91,1] = PR[90,1] + 10.990;
   1:  PR[91,2] = PR[90,2] + 19.933;
   1:L PR[91] R[100]mm/sec CNT100;
   1:  PR[91,1] = PR[90,1] + 8.041;
   1:  PR[91,2] = PR[90,2] + 19.728;
   1:L PR[91] R[100]mm/sec CNT100;
   1:  PR[91,1] = PR[90,1] + 5.891;
   1:  PR[91,2] = PR[90,2] + 19.164;
   1:L PR[91] R[100]mm/sec CNT100;
   1:  PR[91,1] = PR[90,1] + 3.432;
   1:  PR[91,2] = PR[90,2] + 18.445;
   1:L PR[91] R[100]mm/sec CNT100;
   1:  PR[91,1] = PR[90,1] + 3.054;
   1:  PR[91,2] = PR[90,2] + 18.273;
   1:L PR[91] R[100]mm/sec CNT100;
   1:  PR[91,1] = PR[90,1] + 1.377;
   1:  PR[91,2] = PR[90,2] + 17.414;
   1:L PR[91] R[100]mm/sec CNT100;
   1:  PR[91,1] = PR[90,1] + 1.007;
   1:  PR[91,2] = PR[90,2] + 17.317;
   1:L PR[91] R[100]mm/sec CNT100;
   1:  PR[91,1] = PR[90,1] + -0.176;
   1:  PR[91,2] = PR[90,2] + 16.905;
   1:L PR[91] R[100]mm/sec CNT100;
   1:  PR[91] = PR[90];
   1:  PR[91,1] = PR[90,1] + -1.000;
   1:  PR[91,2] = PR[90,2] + 17.682;
   1:  PR[91,3] = PR[90,3] + 44.395;
   1:L PR[91] R[100]mm/sec CNT100;
   1:  PR[91,1] = PR[90,1] + -1.709;
   1:  PR[91,2] = PR[90,2] + 17.789;
   1:L PR[91] R[100]mm/sec CNT100;
   1:  PR[91,1] = PR[90,1] + -2.943;
   1:  PR[91,2] = PR[90,2] + 18.422;
   1:L PR[91] R[100]mm/sec CNT100;
   1:  PR[91,1] = PR[90,1] + -3.443;
   1:  PR[91,2] = PR[90,2] + 18.650;
   1:L PR[91] R[100]mm/sec CNT100;
   1:  PR[91,1] = PR[90,1] + -5.344;
   1:  PR[91,2] = PR[90,2] + 19.206;
   1:L PR[91] R[100]mm/sec CNT100;
   1:  PR[91,1] = PR[90,1] + -8.083;
   1:  PR[91,2] = PR[90,2] + 19.924;
   1:L PR[91] R[100]mm/sec CNT100;
   1:  PR[91,1] = PR[90,1] + -10.453;
   1:  PR[91,2] = PR[90,2] + 20.088;
   1:L PR[91] R[100]mm/sec CNT100;
   1:  PR[91,1] = PR[90,1] + -12.810;
   1:  PR[91,2] = PR[90,2] + 20.185;
   1:L PR[91] R[100]mm/sec CNT100;
   1:  PR[91,1] = PR[90,1] + -15.544;
   1:  PR[91,2] = PR[90,2] + 19.790;
   1:L PR[91] R[100]mm/sec CNT100;
   1:  PR[91,1] = PR[90,1] + -17.487;
   1:  PR[91,2] = PR[90,2] + 19.458;
   1:L PR[91] R[100]mm/sec CNT100;
   1:  PR[91,1] = PR[90,1] + -20.425;
   1:  PR[91,2] = PR[90,2] + 18.368;
   1:L PR[91] R[100]mm/sec CNT100;
   1:  PR[91,1] = PR[90,1] + -21.885;
   1:  PR[91,2] = PR[90,2] + 17.786;
   1:L PR[91] R[100]mm/sec CNT100;
   1:  PR[91,1] = PR[90,1] + -24.807;
   1:  PR[91,2] = PR[90,2] + 15.924;
   1:L PR[91] R[100]mm/sec CNT100;
   1:  PR[91,1] = PR[90,1] + -25.795;
   1:  PR[91,2] = PR[90,2] + 15.263;
   1:L PR[91] R[100]mm/sec CNT100;
   1:  PR[91,1] = PR[90,1] + -28.439;
   1:  PR[91,2] = PR[90,2] + 12.630;
   1:L PR[91] R[100]mm/sec CNT100;
   1:  PR[91,1] = PR[90,1] + -29.032;
   1:  PR[91,2] = PR[90,2] + 12.015;
   1:L PR[91] R[100]mm/sec CNT100;
   1:  PR[91,1] = PR[90,1] + -31.138;
   1:  PR[91,2] = PR[90,2] + 8.686;
   1:L PR[91] R[100]mm/sec CNT100;
   1:  PR[91,1] = PR[90,1] + -31.455;
   1:  PR[91,2] = PR[90,2] + 8.168;
   1:L PR[91] R[100]mm/sec CNT100;
   1:  PR[91,1] = PR[90,1] + -32.951;
   1:  PR[91,2] = PR[90,2] + 4.014;
   1:L PR[91] R[100]mm/sec CNT100;
   1:  PR[91,1] = PR[90,1] + -33.412;
   1:  PR[91,2] = PR[90,2] + -0.035;
   1:L PR[91] R[100]mm/sec CNT100;
   1:  PR[91,1] = PR[90,1] + -33.440;
   1:  PR[91,2] = PR[90,2] + -0.384;
   1:L PR[91] R[100]mm/sec CNT100;
   1:  PR[91,1] = PR[90,1] + -33.094;
   1:  PR[91,2] = PR[90,2] + -3.407;
   1:L PR[91] R[100]mm/sec CNT100;
   1:  PR[91,1] = PR[90,1] + -32.944;
   1:  PR[91,2] = PR[90,2] + -4.888;
   1:L PR[91] R[100]mm/sec CNT100;
   1:  PR[91,1] = PR[90,1] + -32.812;
   1:  PR[91,2] = PR[90,2] + -5.269;
   1:L PR[91] R[100]mm/sec CNT100;
   1:  PR[91,1] = PR[90,1] + -31.456;
   1:  PR[91,2] = PR[90,2] + -9.014;
   1:L PR[91] R[100]mm/sec CNT100;
   1:  PR[91,1] = PR[90,1] + -31.138;
   1:  PR[91,2] = PR[90,2] + -9.533;
   1:L PR[91] R[100]mm/sec CNT100;
   1:  PR[91,1] = PR[90,1] + -29.031;
   1:  PR[91,2] = PR[90,2] + -12.863;
   1:L PR[91] R[100]mm/sec CNT100;
   1:  PR[91,1] = PR[90,1] + -28.439;
   1:  PR[91,2] = PR[90,2] + -13.477;
   1:L PR[91] R[100]mm/sec CNT100;
   1:  PR[91,1] = PR[90,1] + -25.795;
   1:  PR[91,2] = PR[90,2] + -16.110;
   1:L PR[91] R[100]mm/sec CNT100;
   1:  PR[91,1] = PR[90,1] + -24.807;
   1:  PR[91,2] = PR[90,2] + -16.772;
   1:L PR[91] R[100]mm/sec CNT100;
   1:  PR[91,1] = PR[90,1] + -21.885;
   1:  PR[91,2] = PR[90,2] + -18.633;
   1:L PR[91] R[100]mm/sec CNT100;
   1:  PR[91,1] = PR[90,1] + -20.424;
   1:  PR[91,2] = PR[90,2] + -19.215;
   1:L PR[91] R[100]mm/sec CNT100;
   1:  PR[91,1] = PR[90,1] + -17.486;
   1:  PR[91,2] = PR[90,2] + -20.306;
   1:L PR[91] R[100]mm/sec CNT100;
   1:  PR[91,1] = PR[90,1] + -15.544;
   1:  PR[91,2] = PR[90,2] + -20.637;
   1:L PR[91] R[100]mm/sec CNT100;
   1:  PR[91,1] = PR[90,1] + -12.810;
   1:  PR[91,2] = PR[90,2] + -21.032;
   1:L PR[91] R[100]mm/sec CNT100;
   1:  PR[91,1] = PR[90,1] + -10.453;
   1:  PR[91,2] = PR[90,2] + -20.935;
   1:L PR[91] R[100]mm/sec CNT100;
   1:  PR[91,1] = PR[90,1] + -8.083;
   1:  PR[91,2] = PR[90,2] + -20.771;
   1:L PR[91] R[100]mm/sec CNT100;
   1:  PR[91,1] = PR[90,1] + -5.341;
   1:  PR[91,2] = PR[90,2] + -20.052;
   1:L PR[91] R[100]mm/sec CNT100;
   1:  PR[91,1] = PR[90,1] + -3.442;
   1:  PR[91,2] = PR[90,2] + -19.497;
   1:L PR[91] R[100]mm/sec CNT100;
   1:  PR[91,1] = PR[90,1] + -2.904;
   1:  PR[91,2] = PR[90,2] + -19.251;
   1:L PR[91] R[100]mm/sec CNT100;
   1:  PR[91,1] = PR[90,1] + -1.712;
   1:  PR[91,2] = PR[90,2] + -18.638;
   1:L PR[91] R[100]mm/sec CNT100;
   1:  PR[91,1] = PR[90,1] + -0.999;
   1:  PR[91,2] = PR[90,2] + -18.529;
   1:L PR[91] R[100]mm/sec CNT100;
   1:  PR[91,1] = PR[90,1] + -0.134;
   1:  PR[91,2] = PR[90,2] + -18.221;
   1:L PR[91] R[100]mm/sec CNT100;
   1:  PR[91,1] = PR[90,1] + 0.871;
   1:  PR[91,2] = PR[90,2] + -18.572;
   1:L PR[91] R[100]mm/sec CNT100;
   1:  PR[91,1] = PR[90,1] + 1.347;
   1:  PR[91,2] = PR[90,2] + -18.699;
   1:L PR[91] R[100]mm/sec CNT100;
   1:  PR[91,1] = PR[90,1] + 2.420;
   1:  PR[91,2] = PR[90,2] + -19.249;
   1:L PR[91] R[100]mm/sec CNT100;
   1:  PR[91,1] = PR[90,1] + 2.961;
   1:  PR[91,2] = PR[90,2] + -19.495;
   1:L PR[91] R[100]mm/sec CNT100;
   1:  PR[91,1] = PR[90,1] + 4.861;
   1:  PR[91,2] = PR[90,2] + -20.051;
   1:L PR[91] R[100]mm/sec CNT100;
   1:  PR[91,1] = PR[90,1] + 7.602;
   1:  PR[91,2] = PR[90,2] + -20.771;
   1:L PR[91] R[100]mm/sec CNT100;
   1:  PR[91,1] = PR[90,1] + 9.972;
   1:  PR[91,2] = PR[90,2] + -20.935;
   1:L PR[91] R[100]mm/sec CNT100;
   1:  PR[91,1] = PR[90,1] + 12.328;
   1:  PR[91,2] = PR[90,2] + -21.032;
   1:L PR[91] R[100]mm/sec CNT100;
   1:  PR[91,1] = PR[90,1] + 15.062;
   1:  PR[91,2] = PR[90,2] + -20.637;
   1:L PR[91] R[100]mm/sec CNT100;
   1:  PR[91,1] = PR[90,1] + 17.005;
   1:  PR[91,2] = PR[90,2] + -20.305;
   1:L PR[91] R[100]mm/sec CNT100;
   1:  PR[91,1] = PR[90,1] + 19.943;
   1:  PR[91,2] = PR[90,2] + -19.216;
   1:L PR[91] R[100]mm/sec CNT100;
   1:  PR[91,1] = PR[90,1] + 21.405;
   1:  PR[91,2] = PR[90,2] + -18.634;
   1:L PR[91] R[100]mm/sec CNT100;
   1:  PR[91,1] = PR[90,1] + 24.326;
   1:  PR[91,2] = PR[90,2] + -16.775;
   1:L PR[91] R[100]mm/sec CNT100;
   1:  PR[91,1] = PR[90,1] + 25.313;
   1:  PR[91,2] = PR[90,2] + -16.115;
   1:L PR[91] R[100]mm/sec CNT100;
   1:  PR[91,1] = PR[90,1] + 27.957;
   1:  PR[91,2] = PR[90,2] + -13.474;
   1:L PR[91] R[100]mm/sec CNT100;
   1:  PR[91,1] = PR[90,1] + 28.551;
   1:  PR[91,2] = PR[90,2] + -12.857;
   1:L PR[91] R[100]mm/sec CNT100;
   1:  PR[91,1] = PR[90,1] + 30.659;
   1:  PR[91,2] = PR[90,2] + -9.531;
   1:L PR[91] R[100]mm/sec CNT100;
   1:  PR[91,1] = PR[90,1] + 30.976;
   1:  PR[91,2] = PR[90,2] + -9.014;
   1:L PR[91] R[100]mm/sec CNT100;
   1:  PR[91,1] = PR[90,1] + 32.471;
   1:  PR[91,2] = PR[90,2] + -4.878;
   1:L PR[91] R[100]mm/sec CNT100;
   1:  PR[91,1] = PR[90,1] + 32.932;
   1:  PR[91,2] = PR[90,2] + -0.814;
   1:L PR[91] R[100]mm/sec CNT100;
   1:  PR[91,1] = PR[90,1] + 32.960;
   1:  PR[91,2] = PR[90,2] + -0.463;
   1:L PR[91] R[100]mm/sec CNT100;
   1:  PR[91,1] = PR[90,1] + 32.614;
   1:  PR[91,2] = PR[90,2] + 2.573;
   1:L PR[91] R[100]mm/sec CNT100;
   1:  PR[91,1] = PR[90,1] + 32.466;
   1:  PR[91,2] = PR[90,2] + 4.045;
   1:L PR[91] R[100]mm/sec CNT100;
   1:  PR[91,1] = PR[90,1] + 30.976;
   1:  PR[91,2] = PR[90,2] + 8.166;
   1:L PR[91] R[100]mm/sec CNT100;
   1:  PR[91,1] = PR[90,1] + 30.659;
   1:  PR[91,2] = PR[90,2] + 8.684;
   1:L PR[91] R[100]mm/sec CNT100;
   1:  PR[91,1] = PR[90,1] + 28.551;
   1:  PR[91,2] = PR[90,2] + 12.010;
   1:L PR[91] R[100]mm/sec CNT100;
   1:  PR[91,1] = PR[90,1] + 27.957;
   1:  PR[91,2] = PR[90,2] + 12.627;
   1:L PR[91] R[100]mm/sec CNT100;
   1:  PR[91,1] = PR[90,1] + 25.313;
   1:  PR[91,2] = PR[90,2] + 15.268;
   1:L PR[91] R[100]mm/sec CNT100;
   1:  PR[91,1] = PR[90,1] + 24.326;
   1:  PR[91,2] = PR[90,2] + 15.928;
   1:L PR[91] R[100]mm/sec CNT100;
   1:  PR[91,1] = PR[90,1] + 21.405;
   1:  PR[91,2] = PR[90,2] + 17.786;
   1:L PR[91] R[100]mm/sec CNT100;
   1:  PR[91,1] = PR[90,1] + 19.944;
   1:  PR[91,2] = PR[90,2] + 18.368;
   1:L PR[91] R[100]mm/sec CNT100;
   1:  PR[91,1] = PR[90,1] + 17.005;
   1:  PR[91,2] = PR[90,2] + 19.458;
   1:L PR[91] R[100]mm/sec CNT100;
   1:  PR[91,1] = PR[90,1] + 15.062;
   1:  PR[91,2] = PR[90,2] + 19.790;
   1:L PR[91] R[100]mm/sec CNT100;
   1:  PR[91,1] = PR[90,1] + 12.329;
   1:  PR[91,2] = PR[90,2] + 20.185;
   1:L PR[91] R[100]mm/sec CNT100;
   1:  PR[91,1] = PR[90,1] + 9.972;
   1:  PR[91,2] = PR[90,2] + 20.088;
   1:L PR[91] R[100]mm/sec CNT100;
   1:  PR[91,1] = PR[90,1] + 7.602;
   1:  PR[91,2] = PR[90,2] + 19.924;
   1:L PR[91] R[100]mm/sec CNT100;
   1:  PR[91,1] = PR[90,1] + 4.863;
   1:  PR[91,2] = PR[90,2] + 19.205;
   1:L PR[91] R[100]mm/sec CNT100;
   1:  PR[91,1] = PR[90,1] + 2.961;
   1:  PR[91,2] = PR[90,2] + 18.648;
   1:L PR[91] R[100]mm/sec CNT100;
   1:  PR[91,1] = PR[90,1] + 2.460;
   1:  PR[91,2] = PR[90,2] + 18.421;
   1:L PR[91] R[100]mm/sec CNT100;
   1:  PR[91,1] = PR[90,1] + 1.342;
   1:  PR[91,2] = PR[90,2] + 17.848;
   1:L PR[91] R[100]mm/sec CNT100;
   1:  PR[91,1] = PR[90,1] + 0.866;
   1:  PR[91,2] = PR[90,2] + 17.723;
   1:L PR[91] R[100]mm/sec CNT100;
   1:  PR[91,1] = PR[90,1] + -0.135;
   1:  PR[91,2] = PR[90,2] + 17.374;
   1:L PR[91] R[100]mm/sec CNT100;
   1:  PR[91] = PR[90];
   1:  PR[91,1] = PR[90,1] + -0.781;
   1:  PR[91,2] = PR[90,2] + 18.088;
   1:  PR[91,3] = PR[90,3] + 45.695;
   1:L PR[91] R[100]mm/sec CNT100;
   1:  PR[91,1] = PR[90,1] + -1.673;
   1:  PR[91,2] = PR[90,2] + 18.223;
   1:L PR[91] R[100]mm/sec CNT100;
   1:  PR[91,1] = PR[90,1] + -2.350;
   1:  PR[91,2] = PR[90,2] + 18.570;
   1:L PR[91] R[100]mm/sec CNT100;
   1:  PR[91,1] = PR[90,1] + -2.971;
   1:  PR[91,2] = PR[90,2] + 18.853;
   1:L PR[91] R[100]mm/sec CNT100;
   1:  PR[91,1] = PR[90,1] + -4.316;
   1:  PR[91,2] = PR[90,2] + 19.246;
   1:L PR[91] R[100]mm/sec CNT100;
   1:  PR[91,1] = PR[90,1] + -7.645;
   1:  PR[91,2] = PR[90,2] + 20.120;
   1:L PR[91] R[100]mm/sec CNT100;
   1:  PR[91,1] = PR[90,1] + -9.434;
   1:  PR[91,2] = PR[90,2] + 20.243;
   1:L PR[91] R[100]mm/sec CNT100;
   1:  PR[91,1] = PR[90,1] + -12.395;
   1:  PR[91,2] = PR[90,2] + 20.365;
   1:L PR[91] R[100]mm/sec CNT100;
   1:  PR[91,1] = PR[90,1] + -14.537;
   1:  PR[91,2] = PR[90,2] + 20.055;
   1:L PR[91] R[100]mm/sec CNT100;
   1:  PR[91,1] = PR[90,1] + -17.091;
   1:  PR[91,2] = PR[90,2] + 19.619;
   1:L PR[91] R[100]mm/sec CNT100;
   1:  PR[91,1] = PR[90,1] + -19.457;
   1:  PR[91,2] = PR[90,2] + 18.741;
   1:L PR[91] R[100]mm/sec CNT100;
   1:  PR[91,1] = PR[90,1] + -21.505;
   1:  PR[91,2] = PR[90,2] + 17.925;
   1:L PR[91] R[100]mm/sec CNT100;
   1:  PR[91,1] = PR[90,1] + -23.907;
   1:  PR[91,2] = PR[90,2] + 16.395;
   1:L PR[91] R[100]mm/sec CNT100;
   1:  PR[91,1] = PR[90,1] + -25.427;
   1:  PR[91,2] = PR[90,2] + 15.377;
   1:L PR[91] R[100]mm/sec CNT100;
   1:  PR[91,1] = PR[90,1] + -27.634;
   1:  PR[91,2] = PR[90,2] + 13.180;
   1:L PR[91] R[100]mm/sec CNT100;
   1:  PR[91,1] = PR[90,1] + -28.672;
   1:  PR[91,2] = PR[90,2] + 12.103;
   1:L PR[91] R[100]mm/sec CNT100;
   1:  PR[91,1] = PR[90,1] + -30.450;
   1:  PR[91,2] = PR[90,2] + 9.294;
   1:L PR[91] R[100]mm/sec CNT100;
   1:  PR[91,1] = PR[90,1] + -31.104;
   1:  PR[91,2] = PR[90,2] + 8.227;
   1:L PR[91] R[100]mm/sec CNT100;
   1:  PR[91,1] = PR[90,1] + -32.255;
   1:  PR[91,2] = PR[90,2] + 5.047;
   1:L PR[91] R[100]mm/sec CNT100;
   1:  PR[91,1] = PR[90,1] + -32.600;
   1:  PR[91,2] = PR[90,2] + 4.055;
   1:L PR[91] R[100]mm/sec CNT100;
   1:  PR[91,1] = PR[90,1] + -32.994;
   1:  PR[91,2] = PR[90,2] + 0.595;
   1:L PR[91] R[100]mm/sec CNT100;
   1:  PR[91,1] = PR[90,1] + -33.073;
   1:  PR[91,2] = PR[90,2] + -0.384;
   1:L PR[91] R[100]mm/sec CNT100;
   1:  PR[91,1] = PR[90,1] + -32.903;
   1:  PR[91,2] = PR[90,2] + -1.870;
   1:L PR[91] R[100]mm/sec CNT100;
   1:  PR[91,1] = PR[90,1] + -32.711;
   1:  PR[91,2] = PR[90,2] + -3.896;
   1:L PR[91] R[100]mm/sec CNT100;
   1:  PR[91,1] = PR[90,1] + -32.599;
   1:  PR[91,2] = PR[90,2] + -4.905;
   1:L PR[91] R[100]mm/sec CNT100;
   1:  PR[91,1] = PR[90,1] + -32.255;
   1:  PR[91,2] = PR[90,2] + -5.894;
   1:L PR[91] R[100]mm/sec CNT100;
   1:  PR[91,1] = PR[90,1] + -31.104;
   1:  PR[91,2] = PR[90,2] + -9.074;
   1:L PR[91] R[100]mm/sec CNT100;
   1:  PR[91,1] = PR[90,1] + -30.449;
   1:  PR[91,2] = PR[90,2] + -10.142;
   1:L PR[91] R[100]mm/sec CNT100;
   1:  PR[91,1] = PR[90,1] + -28.672;
   1:  PR[91,2] = PR[90,2] + -12.950;
   1:L PR[91] R[100]mm/sec CNT100;
   1:  PR[91,1] = PR[90,1] + -27.633;
   1:  PR[91,2] = PR[90,2] + -14.027;
   1:L PR[91] R[100]mm/sec CNT100;
   1:  PR[91,1] = PR[90,1] + -25.427;
   1:  PR[91,2] = PR[90,2] + -16.225;
   1:L PR[91] R[100]mm/sec CNT100;
   1:  PR[91,1] = PR[90,1] + -23.907;
   1:  PR[91,2] = PR[90,2] + -17.242;
   1:L PR[91] R[100]mm/sec CNT100;
   1:  PR[91,1] = PR[90,1] + -21.505;
   1:  PR[91,2] = PR[90,2] + -18.772;
   1:L PR[91] R[100]mm/sec CNT100;
   1:  PR[91,1] = PR[90,1] + -19.456;
   1:  PR[91,2] = PR[90,2] + -19.589;
   1:L PR[91] R[100]mm/sec CNT100;
   1:  PR[91,1] = PR[90,1] + -17.090;
   1:  PR[91,2] = PR[90,2] + -20.467;
   1:L PR[91] R[100]mm/sec CNT100;
   1:  PR[91,1] = PR[90,1] + -14.537;
   1:  PR[91,2] = PR[90,2] + -20.903;
   1:L PR[91] R[100]mm/sec CNT100;
   1:  PR[91,1] = PR[90,1] + -12.395;
   1:  PR[91,2] = PR[90,2] + -21.212;
   1:L PR[91] R[100]mm/sec CNT100;
   1:  PR[91,1] = PR[90,1] + -9.434;
   1:  PR[91,2] = PR[90,2] + -21.090;
   1:L PR[91] R[100]mm/sec CNT100;
   1:  PR[91,1] = PR[90,1] + -7.645;
   1:  PR[91,2] = PR[90,2] + -20.967;
   1:L PR[91] R[100]mm/sec CNT100;
   1:  PR[91,1] = PR[90,1] + -4.312;
   1:  PR[91,2] = PR[90,2] + -20.092;
   1:L PR[91] R[100]mm/sec CNT100;
   1:  PR[91,1] = PR[90,1] + -2.971;
   1:  PR[91,2] = PR[90,2] + -19.700;
   1:L PR[91] R[100]mm/sec CNT100;
   1:  PR[91,1] = PR[90,1] + -2.303;
   1:  PR[91,2] = PR[90,2] + -19.395;
   1:L PR[91] R[100]mm/sec CNT100;
   1:  PR[91,1] = PR[90,1] + -1.676;
   1:  PR[91,2] = PR[90,2] + -19.073;
   1:L PR[91] R[100]mm/sec CNT100;
   1:  PR[91,1] = PR[90,1] + -0.781;
   1:  PR[91,2] = PR[90,2] + -18.936;
   1:L PR[91] R[100]mm/sec CNT100;
   1:  PR[91,1] = PR[90,1] + -0.167;
   1:  PR[91,2] = PR[90,2] + -18.717;
   1:L PR[91] R[100]mm/sec CNT100;
   1:  PR[91,1] = PR[90,1] + 1.329;
   1:  PR[91,2] = PR[90,2] + -19.142;
   1:L PR[91] R[100]mm/sec CNT100;
   1:  PR[91,1] = PR[90,1] + 1.820;
   1:  PR[91,2] = PR[90,2] + -19.394;
   1:L PR[91] R[100]mm/sec CNT100;
   1:  PR[91,1] = PR[90,1] + 2.490;
   1:  PR[91,2] = PR[90,2] + -19.699;
   1:L PR[91] R[100]mm/sec CNT100;
   1:  PR[91,1] = PR[90,1] + 3.833;
   1:  PR[91,2] = PR[90,2] + -20.092;
   1:L PR[91] R[100]mm/sec CNT100;
   1:  PR[91,1] = PR[90,1] + 7.164;
   1:  PR[91,2] = PR[90,2] + -20.966;
   1:L PR[91] R[100]mm/sec CNT100;
   1:  PR[91,1] = PR[90,1] + 8.954;
   1:  PR[91,2] = PR[90,2] + -21.090;
   1:L PR[91] R[100]mm/sec CNT100;
   1:  PR[91,1] = PR[90,1] + 11.913;
   1:  PR[91,2] = PR[90,2] + -21.212;
   1:L PR[91] R[100]mm/sec CNT100;
   1:  PR[91,1] = PR[90,1] + 14.056;
   1:  PR[91,2] = PR[90,2] + -20.903;
   1:L PR[91] R[100]mm/sec CNT100;
   1:  PR[91,1] = PR[90,1] + 16.609;
   1:  PR[91,2] = PR[90,2] + -20.466;
   1:L PR[91] R[100]mm/sec CNT100;
   1:  PR[91,1] = PR[90,1] + 18.976;
   1:  PR[91,2] = PR[90,2] + -19.589;
   1:L PR[91] R[100]mm/sec CNT100;
   1:  PR[91,1] = PR[90,1] + 21.025;
   1:  PR[91,2] = PR[90,2] + -18.773;
   1:L PR[91] R[100]mm/sec CNT100;
   1:  PR[91,1] = PR[90,1] + 23.427;
   1:  PR[91,2] = PR[90,2] + -17.244;
   1:L PR[91] R[100]mm/sec CNT100;
   1:  PR[91,1] = PR[90,1] + 24.945;
   1:  PR[91,2] = PR[90,2] + -16.229;
   1:L PR[91] R[100]mm/sec CNT100;
   1:  PR[91,1] = PR[90,1] + 27.151;
   1:  PR[91,2] = PR[90,2] + -14.026;
   1:L PR[91] R[100]mm/sec CNT100;
   1:  PR[91,1] = PR[90,1] + 28.192;
   1:  PR[91,2] = PR[90,2] + -12.945;
   1:L PR[91] R[100]mm/sec CNT100;
   1:  PR[91,1] = PR[90,1] + 29.970;
   1:  PR[91,2] = PR[90,2] + -10.139;
   1:L PR[91] R[100]mm/sec CNT100;
   1:  PR[91,1] = PR[90,1] + 30.625;
   1:  PR[91,2] = PR[90,2] + -9.072;
   1:L PR[91] R[100]mm/sec CNT100;
   1:  PR[91,1] = PR[90,1] + 31.775;
   1:  PR[91,2] = PR[90,2] + -5.905;
   1:L PR[91] R[100]mm/sec CNT100;
   1:  PR[91,1] = PR[90,1] + 32.120;
   1:  PR[91,2] = PR[90,2] + -4.918;
   1:L PR[91] R[100]mm/sec CNT100;
   1:  PR[91,1] = PR[90,1] + 32.514;
   1:  PR[91,2] = PR[90,2] + -1.446;
   1:L PR[91] R[100]mm/sec CNT100;
   1:  PR[91,1] = PR[90,1] + 32.593;
   1:  PR[91,2] = PR[90,2] + -0.463;
   1:L PR[91] R[100]mm/sec CNT100;
   1:  PR[91,1] = PR[90,1] + 32.423;
   1:  PR[91,2] = PR[90,2] + 1.030;
   1:L PR[91] R[100]mm/sec CNT100;
   1:  PR[91,1] = PR[90,1] + 32.231;
   1:  PR[91,2] = PR[90,2] + 3.064;
   1:L PR[91] R[100]mm/sec CNT100;
   1:  PR[91,1] = PR[90,1] + 32.119;
   1:  PR[91,2] = PR[90,2] + 4.074;
   1:L PR[91] R[100]mm/sec CNT100;
   1:  PR[91,1] = PR[90,1] + 31.775;
   1:  PR[91,2] = PR[90,2] + 5.058;
   1:L PR[91] R[100]mm/sec CNT100;
   1:  PR[91,1] = PR[90,1] + 30.625;
   1:  PR[91,2] = PR[90,2] + 8.225;
   1:L PR[91] R[100]mm/sec CNT100;
   1:  PR[91,1] = PR[90,1] + 29.970;
   1:  PR[91,2] = PR[90,2] + 9.292;
   1:L PR[91] R[100]mm/sec CNT100;
   1:  PR[91,1] = PR[90,1] + 28.192;
   1:  PR[91,2] = PR[90,2] + 12.098;
   1:L PR[91] R[100]mm/sec CNT100;
   1:  PR[91,1] = PR[90,1] + 27.151;
   1:  PR[91,2] = PR[90,2] + 13.178;
   1:L PR[91] R[100]mm/sec CNT100;
   1:  PR[91,1] = PR[90,1] + 24.945;
   1:  PR[91,2] = PR[90,2] + 15.382;
   1:L PR[91] R[100]mm/sec CNT100;
   1:  PR[91,1] = PR[90,1] + 23.427;
   1:  PR[91,2] = PR[90,2] + 16.397;
   1:L PR[91] R[100]mm/sec CNT100;
   1:  PR[91,1] = PR[90,1] + 21.025;
   1:  PR[91,2] = PR[90,2] + 17.925;
   1:L PR[91] R[100]mm/sec CNT100;
   1:  PR[91,1] = PR[90,1] + 18.976;
   1:  PR[91,2] = PR[90,2] + 18.741;
   1:L PR[91] R[100]mm/sec CNT100;
   1:  PR[91,1] = PR[90,1] + 16.610;
   1:  PR[91,2] = PR[90,2] + 19.619;
   1:L PR[91] R[100]mm/sec CNT100;
   1:  PR[91,1] = PR[90,1] + 14.056;
   1:  PR[91,2] = PR[90,2] + 20.056;
   1:L PR[91] R[100]mm/sec CNT100;
   1:  PR[91,1] = PR[90,1] + 11.914;
   1:  PR[91,2] = PR[90,2] + 20.365;
   1:L PR[91] R[100]mm/sec CNT100;
   1:  PR[91,1] = PR[90,1] + 8.954;
   1:  PR[91,2] = PR[90,2] + 20.243;
   1:L PR[91] R[100]mm/sec CNT100;
   1:  PR[91,1] = PR[90,1] + 7.164;
   1:  PR[91,2] = PR[90,2] + 20.119;
   1:L PR[91] R[100]mm/sec CNT100;
   1:  PR[91,1] = PR[90,1] + 3.836;
   1:  PR[91,2] = PR[90,2] + 19.246;
   1:L PR[91] R[100]mm/sec CNT100;
   1:  PR[91,1] = PR[90,1] + 2.491;
   1:  PR[91,2] = PR[90,2] + 18.852;
   1:L PR[91] R[100]mm/sec CNT100;
   1:  PR[91,1] = PR[90,1] + 1.867;
   1:  PR[91,2] = PR[90,2] + 18.569;
   1:L PR[91] R[100]mm/sec CNT100;
   1:  PR[91,1] = PR[90,1] + 1.325;
   1:  PR[91,2] = PR[90,2] + 18.291;
   1:L PR[91] R[100]mm/sec CNT100;
   1:  PR[91,1] = PR[90,1] + -0.172;
   1:  PR[91,2] = PR[90,2] + 17.871;
   1:L PR[91] R[100]mm/sec CNT100;
   1:  PR[91] = PR[90];
   1:  PR[91,1] = PR[90,1] + -1.582;
   1:  PR[91,2] = PR[90,2] + 18.639;
   1:  PR[91,3] = PR[90,3] + 46.995;
   1:L PR[91] R[100]mm/sec CNT100;
   1:  PR[91,1] = PR[90,1] + -2.500;
   1:  PR[91,2] = PR[90,2] + 19.057;
   1:L PR[91] R[100]mm/sec CNT100;
   1:  PR[91,1] = PR[90,1] + -3.287;
   1:  PR[91,2] = PR[90,2] + 19.287;
   1:L PR[91] R[100]mm/sec CNT100;
   1:  PR[91,1] = PR[90,1] + -7.206;
   1:  PR[91,2] = PR[90,2] + 20.315;
   1:L PR[91] R[100]mm/sec CNT100;
   1:  PR[91,1] = PR[90,1] + -8.415;
   1:  PR[91,2] = PR[90,2] + 20.398;
   1:L PR[91] R[100]mm/sec CNT100;
   1:  PR[91,1] = PR[90,1] + -11.979;
   1:  PR[91,2] = PR[90,2] + 20.545;
   1:L PR[91] R[100]mm/sec CNT100;
   1:  PR[91,1] = PR[90,1] + -13.531;
   1:  PR[91,2] = PR[90,2] + 20.321;
   1:L PR[91] R[100]mm/sec CNT100;
   1:  PR[91,1] = PR[90,1] + -16.695;
   1:  PR[91,2] = PR[90,2] + 19.781;
   1:L PR[91] R[100]mm/sec CNT100;
   1:  PR[91,1] = PR[90,1] + -18.489;
   1:  PR[91,2] = PR[90,2] + 19.115;
   1:L PR[91] R[100]mm/sec CNT100;
   1:  PR[91,1] = PR[90,1] + -21.125;
   1:  PR[91,2] = PR[90,2] + 18.064;
   1:L PR[91] R[100]mm/sec CNT100;
   1:  PR[91,1] = PR[90,1] + -23.007;
   1:  PR[91,2] = PR[90,2] + 16.865;
   1:L PR[91] R[100]mm/sec CNT100;
   1:  PR[91,1] = PR[90,1] + -25.059;
   1:  PR[91,2] = PR[90,2] + 15.492;
   1:L PR[91] R[100]mm/sec CNT100;
   1:  PR[91,1] = PR[90,1] + -26.828;
   1:  PR[91,2] = PR[90,2] + 13.730;
   1:L PR[91] R[100]mm/sec CNT100;
   1:  PR[91,1] = PR[90,1] + -28.313;
   1:  PR[91,2] = PR[90,2] + 12.191;
   1:L PR[91] R[100]mm/sec CNT100;
   1:  PR[91,1] = PR[90,1] + -29.760;
   1:  PR[91,2] = PR[90,2] + 9.904;
   1:L PR[91] R[100]mm/sec CNT100;
   1:  PR[91,1] = PR[90,1] + -30.751;
   1:  PR[91,2] = PR[90,2] + 8.288;
   1:L PR[91] R[100]mm/sec CNT100;
   1:  PR[91,1] = PR[90,1] + -31.698;
   1:  PR[91,2] = PR[90,2] + 5.670;
   1:L PR[91] R[100]mm/sec CNT100;
   1:  PR[91,1] = PR[90,1] + -32.251;
   1:  PR[91,2] = PR[90,2] + 4.082;
   1:L PR[91] R[100]mm/sec CNT100;
   1:  PR[91,1] = PR[90,1] + -32.576;
   1:  PR[91,2] = PR[90,2] + 1.226;
   1:L PR[91] R[100]mm/sec CNT100;
   1:  PR[91,1] = PR[90,1] + -32.708;
   1:  PR[91,2] = PR[90,2] + -0.406;
   1:L PR[91] R[100]mm/sec CNT100;
   1:  PR[91,1] = PR[90,1] + -32.430;
   1:  PR[91,2] = PR[90,2] + -3.309;
   1:L PR[91] R[100]mm/sec CNT100;
   1:  PR[91,1] = PR[90,1] + -32.249;
   1:  PR[91,2] = PR[90,2] + -4.933;
   1:L PR[91] R[100]mm/sec CNT100;
   1:  PR[91,1] = PR[90,1] + -31.698;
   1:  PR[91,2] = PR[90,2] + -6.517;
   1:L PR[91] R[100]mm/sec CNT100;
   1:  PR[91,1] = PR[90,1] + -30.751;
   1:  PR[91,2] = PR[90,2] + -9.135;
   1:L PR[91] R[100]mm/sec CNT100;
   1:  PR[91,1] = PR[90,1] + -29.760;
   1:  PR[91,2] = PR[90,2] + -10.751;
   1:L PR[91] R[100]mm/sec CNT100;
   1:  PR[91,1] = PR[90,1] + -28.313;
   1:  PR[91,2] = PR[90,2] + -13.038;
   1:L PR[91] R[100]mm/sec CNT100;
   1:  PR[91,1] = PR[90,1] + -26.828;
   1:  PR[91,2] = PR[90,2] + -14.578;
   1:L PR[91] R[100]mm/sec CNT100;
   1:  PR[91,1] = PR[90,1] + -25.059;
   1:  PR[91,2] = PR[90,2] + -16.339;
   1:L PR[91] R[100]mm/sec CNT100;
   1:  PR[91,1] = PR[90,1] + -23.007;
   1:  PR[91,2] = PR[90,2] + -17.712;
   1:L PR[91] R[100]mm/sec CNT100;
   1:  PR[91,1] = PR[90,1] + -21.124;
   1:  PR[91,2] = PR[90,2] + -18.912;
   1:L PR[91] R[100]mm/sec CNT100;
   1:  PR[91,1] = PR[90,1] + -18.489;
   1:  PR[91,2] = PR[90,2] + -19.962;
   1:L PR[91] R[100]mm/sec CNT100;
   1:  PR[91,1] = PR[90,1] + -16.694;
   1:  PR[91,2] = PR[90,2] + -20.628;
   1:L PR[91] R[100]mm/sec CNT100;
   1:  PR[91,1] = PR[90,1] + -13.530;
   1:  PR[91,2] = PR[90,2] + -21.168;
   1:L PR[91] R[100]mm/sec CNT100;
   1:  PR[91,1] = PR[90,1] + -11.979;
   1:  PR[91,2] = PR[90,2] + -21.392;
   1:L PR[91] R[100]mm/sec CNT100;
   1:  PR[91,1] = PR[90,1] + -8.415;
   1:  PR[91,2] = PR[90,2] + -21.245;
   1:L PR[91] R[100]mm/sec CNT100;
   1:  PR[91,1] = PR[90,1] + -7.206;
   1:  PR[91,2] = PR[90,2] + -21.162;
   1:L PR[91] R[100]mm/sec CNT100;
   1:  PR[91,1] = PR[90,1] + -3.284;
   1:  PR[91,2] = PR[90,2] + -20.133;
   1:L PR[91] R[100]mm/sec CNT100;
   1:  PR[91,1] = PR[90,1] + -2.499;
   1:  PR[91,2] = PR[90,2] + -19.904;
   1:L PR[91] R[100]mm/sec CNT100;
   1:  PR[91,1] = PR[90,1] + -1.582;
   1:  PR[91,2] = PR[90,2] + -19.485;
   1:L PR[91] R[100]mm/sec CNT100;
   1:  PR[91,1] = PR[90,1] + 0.104;
   1:  PR[91,2] = PR[90,2] + -19.229;
   1:L PR[91] R[100]mm/sec CNT100;
   1:  PR[91,1] = PR[90,1] + 1.236;
   1:  PR[91,2] = PR[90,2] + -19.546;
   1:L PR[91] R[100]mm/sec CNT100;
   1:  PR[91,1] = PR[90,1] + 2.019;
   1:  PR[91,2] = PR[90,2] + -19.903;
   1:L PR[91] R[100]mm/sec CNT100;
   1:  PR[91,1] = PR[90,1] + 2.805;
   1:  PR[91,2] = PR[90,2] + -20.133;
   1:L PR[91] R[100]mm/sec CNT100;
   1:  PR[91,1] = PR[90,1] + 6.726;
   1:  PR[91,2] = PR[90,2] + -21.162;
   1:L PR[91] R[100]mm/sec CNT100;
   1:  PR[91,1] = PR[90,1] + 7.935;
   1:  PR[91,2] = PR[90,2] + -21.246;
   1:L PR[91] R[100]mm/sec CNT100;
   1:  PR[91,1] = PR[90,1] + 11.499;
   1:  PR[91,2] = PR[90,2] + -21.393;
   1:L PR[91] R[100]mm/sec CNT100;
   1:  PR[91,1] = PR[90,1] + 13.050;
   1:  PR[91,2] = PR[90,2] + -21.168;
   1:L PR[91] R[100]mm/sec CNT100;
   1:  PR[91,1] = PR[90,1] + 16.214;
   1:  PR[91,2] = PR[90,2] + -20.627;
   1:L PR[91] R[100]mm/sec CNT100;
   1:  PR[91,1] = PR[90,1] + 18.009;
   1:  PR[91,2] = PR[90,2] + -19.962;
   1:L PR[91] R[100]mm/sec CNT100;
   1:  PR[91,1] = PR[90,1] + 20.645;
   1:  PR[91,2] = PR[90,2] + -18.912;
   1:L PR[91] R[100]mm/sec CNT100;
   1:  PR[91,1] = PR[90,1] + 22.527;
   1:  PR[91,2] = PR[90,2] + -17.714;
   1:L PR[91] R[100]mm/sec CNT100;
   1:  PR[91,1] = PR[90,1] + 24.577;
   1:  PR[91,2] = PR[90,2] + -16.343;
   1:L PR[91] R[100]mm/sec CNT100;
   1:  PR[91,1] = PR[90,1] + 26.346;
   1:  PR[91,2] = PR[90,2] + -14.577;
   1:L PR[91] R[100]mm/sec CNT100;
   1:  PR[91,1] = PR[90,1] + 27.833;
   1:  PR[91,2] = PR[90,2] + -13.033;
   1:L PR[91] R[100]mm/sec CNT100;
   1:  PR[91,1] = PR[90,1] + 29.281;
   1:  PR[91,2] = PR[90,2] + -10.747;
   1:L PR[91] R[100]mm/sec CNT100;
   1:  PR[91,1] = PR[90,1] + 30.272;
   1:  PR[91,2] = PR[90,2] + -9.133;
   1:L PR[91] R[100]mm/sec CNT100;
   1:  PR[91,1] = PR[90,1] + 31.219;
   1:  PR[91,2] = PR[90,2] + -6.526;
   1:L PR[91] R[100]mm/sec CNT100;
   1:  PR[91,1] = PR[90,1] + 31.770;
   1:  PR[91,2] = PR[90,2] + -4.945;
   1:L PR[91] R[100]mm/sec CNT100;
   1:  PR[91,1] = PR[90,1] + 32.096;
   1:  PR[91,2] = PR[90,2] + -2.078;
   1:L PR[91] R[100]mm/sec CNT100;
   1:  PR[91,1] = PR[90,1] + 32.228;
   1:  PR[91,2] = PR[90,2] + -0.441;
   1:L PR[91] R[100]mm/sec CNT100;
   1:  PR[91,1] = PR[90,1] + 31.950;
   1:  PR[91,2] = PR[90,2] + 2.474;
   1:L PR[91] R[100]mm/sec CNT100;
   1:  PR[91,1] = PR[90,1] + 31.769;
   1:  PR[91,2] = PR[90,2] + 4.101;
   1:L PR[91] R[100]mm/sec CNT100;
   1:  PR[91,1] = PR[90,1] + 31.219;
   1:  PR[91,2] = PR[90,2] + 5.679;
   1:L PR[91] R[100]mm/sec CNT100;
   1:  PR[91,1] = PR[90,1] + 30.272;
   1:  PR[91,2] = PR[90,2] + 8.285;
   1:L PR[91] R[100]mm/sec CNT100;
   1:  PR[91,1] = PR[90,1] + 29.282;
   1:  PR[91,2] = PR[90,2] + 9.899;
   1:L PR[91] R[100]mm/sec CNT100;
   1:  PR[91,1] = PR[90,1] + 27.833;
   1:  PR[91,2] = PR[90,2] + 12.185;
   1:L PR[91] R[100]mm/sec CNT100;
   1:  PR[91,1] = PR[90,1] + 26.346;
   1:  PR[91,2] = PR[90,2] + 13.730;
   1:L PR[91] R[100]mm/sec CNT100;
   1:  PR[91,1] = PR[90,1] + 24.577;
   1:  PR[91,2] = PR[90,2] + 15.496;
   1:L PR[91] R[100]mm/sec CNT100;
   1:  PR[91,1] = PR[90,1] + 22.527;
   1:  PR[91,2] = PR[90,2] + 16.867;
   1:L PR[91] R[100]mm/sec CNT100;
   1:  PR[91,1] = PR[90,1] + 20.645;
   1:  PR[91,2] = PR[90,2] + 18.065;
   1:L PR[91] R[100]mm/sec CNT100;
   1:  PR[91,1] = PR[90,1] + 18.009;
   1:  PR[91,2] = PR[90,2] + 19.115;
   1:L PR[91] R[100]mm/sec CNT100;
   1:  PR[91,1] = PR[90,1] + 16.214;
   1:  PR[91,2] = PR[90,2] + 19.780;
   1:L PR[91] R[100]mm/sec CNT100;
   1:  PR[91,1] = PR[90,1] + 13.049;
   1:  PR[91,2] = PR[90,2] + 20.321;
   1:L PR[91] R[100]mm/sec CNT100;
   1:  PR[91,1] = PR[90,1] + 11.499;
   1:  PR[91,2] = PR[90,2] + 20.545;
   1:L PR[91] R[100]mm/sec CNT100;
   1:  PR[91,1] = PR[90,1] + 7.935;
   1:  PR[91,2] = PR[90,2] + 20.398;
   1:L PR[91] R[100]mm/sec CNT100;
   1:  PR[91,1] = PR[90,1] + 6.726;
   1:  PR[91,2] = PR[90,2] + 20.315;
   1:L PR[91] R[100]mm/sec CNT100;
   1:  PR[91,1] = PR[90,1] + 2.808;
   1:  PR[91,2] = PR[90,2] + 19.286;
   1:L PR[91] R[100]mm/sec CNT100;
   1:  PR[91,1] = PR[90,1] + 2.020;
   1:  PR[91,2] = PR[90,2] + 19.056;
   1:L PR[91] R[100]mm/sec CNT100;
   1:  PR[91,1] = PR[90,1] + 1.237;
   1:  PR[91,2] = PR[90,2] + 18.700;
   1:L PR[91] R[100]mm/sec CNT100;
   1:  PR[91,1] = PR[90,1] + 0.103;
   1:  PR[91,2] = PR[90,2] + 18.381;
   1:L PR[91] R[100]mm/sec CNT100;
   1:  PR[91] = PR[90];
   1:  PR[91,1] = PR[90,1] + -0.436;
   1:  PR[91,2] = PR[90,2] + 18.844;
   1:  PR[91,3] = PR[90,3] + 48.295;
   1:L PR[91] R[100]mm/sec CNT100;
   1:  PR[91,1] = PR[90,1] + -1.583;
   1:  PR[91,2] = PR[90,2] + 19.057;
   1:L PR[91] R[100]mm/sec CNT100;
   1:  PR[91,1] = PR[90,1] + -2.028;
   1:  PR[91,2] = PR[90,2] + 19.260;
   1:L PR[91] R[100]mm/sec CNT100;
   1:  PR[91,1] = PR[90,1] + -2.259;
   1:  PR[91,2] = PR[90,2] + 19.327;
   1:L PR[91] R[100]mm/sec CNT100;
   1:  PR[91,1] = PR[90,1] + -6.768;
   1:  PR[91,2] = PR[90,2] + 20.510;
   1:L PR[91] R[100]mm/sec CNT100;
   1:  PR[91,1] = PR[90,1] + -7.396;
   1:  PR[91,2] = PR[90,2] + 20.554;
   1:L PR[91] R[100]mm/sec CNT100;
   1:  PR[91,1] = PR[90,1] + -11.564;
   1:  PR[91,2] = PR[90,2] + 20.725;
   1:L PR[91] R[100]mm/sec CNT100;
   1:  PR[91,1] = PR[90,1] + -12.524;
   1:  PR[91,2] = PR[90,2] + 20.587;
   1:L PR[91] R[100]mm/sec CNT100;
   1:  PR[91,1] = PR[90,1] + -16.299;
   1:  PR[91,2] = PR[90,2] + 19.942;
   1:L PR[91] R[100]mm/sec CNT100;
   1:  PR[91,1] = PR[90,1] + -17.522;
   1:  PR[91,2] = PR[90,2] + 19.488;
   1:L PR[91] R[100]mm/sec CNT100;
   1:  PR[91,1] = PR[90,1] + -20.744;
   1:  PR[91,2] = PR[90,2] + 18.204;
   1:L PR[91] R[100]mm/sec CNT100;
   1:  PR[91,1] = PR[90,1] + -22.107;
   1:  PR[91,2] = PR[90,2] + 17.336;
   1:L PR[91] R[100]mm/sec CNT100;
   1:  PR[91,1] = PR[90,1] + -24.691;
   1:  PR[91,2] = PR[90,2] + 15.607;
   1:L PR[91] R[100]mm/sec CNT100;
   1:  PR[91,1] = PR[90,1] + -26.023;
   1:  PR[91,2] = PR[90,2] + 14.280;
   1:L PR[91] R[100]mm/sec CNT100;
   1:  PR[91,1] = PR[90,1] + -27.954;
   1:  PR[91,2] = PR[90,2] + 12.278;
   1:L PR[91] R[100]mm/sec CNT100;
   1:  PR[91,1] = PR[90,1] + -29.072;
   1:  PR[91,2] = PR[90,2] + 10.512;
   1:L PR[91] R[100]mm/sec CNT100;
   1:  PR[91,1] = PR[90,1] + -30.398;
   1:  PR[91,2] = PR[90,2] + 8.348;
   1:L PR[91] R[100]mm/sec CNT100;
   1:  PR[91,1] = PR[90,1] + -31.141;
   1:  PR[91,2] = PR[90,2] + 6.294;
   1:L PR[91] R[100]mm/sec CNT100;
   1:  PR[91,1] = PR[90,1] + -31.901;
   1:  PR[91,2] = PR[90,2] + 4.110;
   1:L PR[91] R[100]mm/sec CNT100;
   1:  PR[91,1] = PR[90,1] + -32.158;
   1:  PR[91,2] = PR[90,2] + 1.857;
   1:L PR[91] R[100]mm/sec CNT100;
   1:  PR[91,1] = PR[90,1] + -32.287;
   1:  PR[91,2] = PR[90,2] + 0.257;
   1:L PR[91] R[100]mm/sec CNT100;
   1:  PR[91,1] = PR[90,1] + -32.365;
   1:  PR[91,2] = PR[90,2] + -0.443;
   1:L PR[91] R[100]mm/sec CNT100;
   1:  PR[91,1] = PR[90,1] + -32.149;
   1:  PR[91,2] = PR[90,2] + -2.723;
   1:L PR[91] R[100]mm/sec CNT100;
   1:  PR[91,1] = PR[90,1] + -31.900;
   1:  PR[91,2] = PR[90,2] + -4.961;
   1:L PR[91] R[100]mm/sec CNT100;
   1:  PR[91,1] = PR[90,1] + -31.141;
   1:  PR[91,2] = PR[90,2] + -7.142;
   1:L PR[91] R[100]mm/sec CNT100;
   1:  PR[91,1] = PR[90,1] + -30.398;
   1:  PR[91,2] = PR[90,2] + -9.195;
   1:L PR[91] R[100]mm/sec CNT100;
   1:  PR[91,1] = PR[90,1] + -29.072;
   1:  PR[91,2] = PR[90,2] + -11.360;
   1:L PR[91] R[100]mm/sec CNT100;
   1:  PR[91,1] = PR[90,1] + -27.954;
   1:  PR[91,2] = PR[90,2] + -13.125;
   1:L PR[91] R[100]mm/sec CNT100;
   1:  PR[91,1] = PR[90,1] + -26.022;
   1:  PR[91,2] = PR[90,2] + -15.128;
   1:L PR[91] R[100]mm/sec CNT100;
   1:  PR[91,1] = PR[90,1] + -24.691;
   1:  PR[91,2] = PR[90,2] + -16.454;
   1:L PR[91] R[100]mm/sec CNT100;
   1:  PR[91,1] = PR[90,1] + -22.107;
   1:  PR[91,2] = PR[90,2] + -18.183;
   1:L PR[91] R[100]mm/sec CNT100;
   1:  PR[91,1] = PR[90,1] + -20.744;
   1:  PR[91,2] = PR[90,2] + -19.051;
   1:L PR[91] R[100]mm/sec CNT100;
   1:  PR[91,1] = PR[90,1] + -17.521;
   1:  PR[91,2] = PR[90,2] + -20.336;
   1:L PR[91] R[100]mm/sec CNT100;
   1:  PR[91,1] = PR[90,1] + -16.298;
   1:  PR[91,2] = PR[90,2] + -20.789;
   1:L PR[91] R[100]mm/sec CNT100;
   1:  PR[91,1] = PR[90,1] + -12.523;
   1:  PR[91,2] = PR[90,2] + -21.434;
   1:L PR[91] R[100]mm/sec CNT100;
   1:  PR[91,1] = PR[90,1] + -11.564;
   1:  PR[91,2] = PR[90,2] + -21.572;
   1:L PR[91] R[100]mm/sec CNT100;
   1:  PR[91,1] = PR[90,1] + -7.396;
   1:  PR[91,2] = PR[90,2] + -21.401;
   1:L PR[91] R[100]mm/sec CNT100;
   1:  PR[91,1] = PR[90,1] + -6.768;
   1:  PR[91,2] = PR[90,2] + -21.357;
   1:L PR[91] R[100]mm/sec CNT100;
   1:  PR[91,1] = PR[90,1] + -2.255;
   1:  PR[91,2] = PR[90,2] + -20.173;
   1:L PR[91] R[100]mm/sec CNT100;
   1:  PR[91,1] = PR[90,1] + -2.028;
   1:  PR[91,2] = PR[90,2] + -20.107;
   1:L PR[91] R[100]mm/sec CNT100;
   1:  PR[91,1] = PR[90,1] + -1.545;
   1:  PR[91,2] = PR[90,2] + -19.887;
   1:L PR[91] R[100]mm/sec CNT100;
   1:  PR[91,1] = PR[90,1] + 0.249;
   1:  PR[91,2] = PR[90,2] + -19.617;
   1:L PR[91] R[100]mm/sec CNT100;
   1:  PR[91,1] = PR[90,1] + 0.937;
   1:  PR[91,2] = PR[90,2] + -19.875;
   1:L PR[91] R[100]mm/sec CNT100;
   1:  PR[91,1] = PR[90,1] + 1.187;
   1:  PR[91,2] = PR[90,2] + -19.942;
   1:L PR[91] R[100]mm/sec CNT100;
   1:  PR[91,1] = PR[90,1] + 1.549;
   1:  PR[91,2] = PR[90,2] + -20.106;
   1:L PR[91] R[100]mm/sec CNT100;
   1:  PR[91,1] = PR[90,1] + 1.777;
   1:  PR[91,2] = PR[90,2] + -20.173;
   1:L PR[91] R[100]mm/sec CNT100;
   1:  PR[91,1] = PR[90,1] + 6.288;
   1:  PR[91,2] = PR[90,2] + -21.357;
   1:L PR[91] R[100]mm/sec CNT100;
   1:  PR[91,1] = PR[90,1] + 6.917;
   1:  PR[91,2] = PR[90,2] + -21.401;
   1:L PR[91] R[100]mm/sec CNT100;
   1:  PR[91,1] = PR[90,1] + 11.084;
   1:  PR[91,2] = PR[90,2] + -21.573;
   1:L PR[91] R[100]mm/sec CNT100;
   1:  PR[91,1] = PR[90,1] + 12.043;
   1:  PR[91,2] = PR[90,2] + -21.434;
   1:L PR[91] R[100]mm/sec CNT100;
   1:  PR[91,1] = PR[90,1] + 15.818;
   1:  PR[91,2] = PR[90,2] + -20.789;
   1:L PR[91] R[100]mm/sec CNT100;
   1:  PR[91,1] = PR[90,1] + 17.042;
   1:  PR[91,2] = PR[90,2] + -20.335;
   1:L PR[91] R[100]mm/sec CNT100;
   1:  PR[91,1] = PR[90,1] + 20.265;
   1:  PR[91,2] = PR[90,2] + -19.051;
   1:L PR[91] R[100]mm/sec CNT100;
   1:  PR[91,1] = PR[90,1] + 21.628;
   1:  PR[91,2] = PR[90,2] + -18.184;
   1:L PR[91] R[100]mm/sec CNT100;
   1:  PR[91,1] = PR[90,1] + 24.209;
   1:  PR[91,2] = PR[90,2] + -16.458;
   1:L PR[91] R[100]mm/sec CNT100;
   1:  PR[91,1] = PR[90,1] + 25.541;
   1:  PR[91,2] = PR[90,2] + -15.128;
   1:L PR[91] R[100]mm/sec CNT100;
   1:  PR[91,1] = PR[90,1] + 27.474;
   1:  PR[91,2] = PR[90,2] + -13.120;
   1:L PR[91] R[100]mm/sec CNT100;
   1:  PR[91,1] = PR[90,1] + 28.593;
   1:  PR[91,2] = PR[90,2] + -11.355;
   1:L PR[91] R[100]mm/sec CNT100;
   1:  PR[91,1] = PR[90,1] + 29.919;
   1:  PR[91,2] = PR[90,2] + -9.193;
   1:L PR[91] R[100]mm/sec CNT100;
   1:  PR[91,1] = PR[90,1] + 30.662;
   1:  PR[91,2] = PR[90,2] + -7.148;
   1:L PR[91] R[100]mm/sec CNT100;
   1:  PR[91,1] = PR[90,1] + 31.421;
   1:  PR[91,2] = PR[90,2] + -4.972;
   1:L PR[91] R[100]mm/sec CNT100;
   1:  PR[91,1] = PR[90,1] + 31.678;
   1:  PR[91,2] = PR[90,2] + -2.710;
   1:L PR[91] R[100]mm/sec CNT100;
   1:  PR[91,1] = PR[90,1] + 31.808;
   1:  PR[91,2] = PR[90,2] + -1.106;
   1:L PR[91] R[100]mm/sec CNT100;
   1:  PR[91,1] = PR[90,1] + 31.885;
   1:  PR[91,2] = PR[90,2] + -0.404;
   1:L PR[91] R[100]mm/sec CNT100;
   1:  PR[91,1] = PR[90,1] + 31.669;
   1:  PR[91,2] = PR[90,2] + 1.887;
   1:L PR[91] R[100]mm/sec CNT100;
   1:  PR[91,1] = PR[90,1] + 31.420;
   1:  PR[91,2] = PR[90,2] + 4.127;
   1:L PR[91] R[100]mm/sec CNT100;
   1:  PR[91,1] = PR[90,1] + 30.662;
   1:  PR[91,2] = PR[90,2] + 6.301;
   1:L PR[91] R[100]mm/sec CNT100;
   1:  PR[91,1] = PR[90,1] + 29.919;
   1:  PR[91,2] = PR[90,2] + 8.346;
   1:L PR[91] R[100]mm/sec CNT100;
   1:  PR[91,1] = PR[90,1] + 28.593;
   1:  PR[91,2] = PR[90,2] + 10.508;
   1:L PR[91] R[100]mm/sec CNT100;
   1:  PR[91,1] = PR[90,1] + 27.474;
   1:  PR[91,2] = PR[90,2] + 12.273;
   1:L PR[91] R[100]mm/sec CNT100;
   1:  PR[91,1] = PR[90,1] + 25.541;
   1:  PR[91,2] = PR[90,2] + 14.281;
   1:L PR[91] R[100]mm/sec CNT100;
   1:  PR[91,1] = PR[90,1] + 24.209;
   1:  PR[91,2] = PR[90,2] + 15.610;
   1:L PR[91] R[100]mm/sec CNT100;
   1:  PR[91,1] = PR[90,1] + 21.628;
   1:  PR[91,2] = PR[90,2] + 17.337;
   1:L PR[91] R[100]mm/sec CNT100;
   1:  PR[91,1] = PR[90,1] + 20.265;
   1:  PR[91,2] = PR[90,2] + 18.204;
   1:L PR[91] R[100]mm/sec CNT100;
   1:  PR[91,1] = PR[90,1] + 17.042;
   1:  PR[91,2] = PR[90,2] + 19.488;
   1:L PR[91] R[100]mm/sec CNT100;
   1:  PR[91,1] = PR[90,1] + 15.818;
   1:  PR[91,2] = PR[90,2] + 19.941;
   1:L PR[91] R[100]mm/sec CNT100;
   1:  PR[91,1] = PR[90,1] + 12.043;
   1:  PR[91,2] = PR[90,2] + 20.587;
   1:L PR[91] R[100]mm/sec CNT100;
   1:  PR[91,1] = PR[90,1] + 11.084;
   1:  PR[91,2] = PR[90,2] + 20.725;
   1:L PR[91] R[100]mm/sec CNT100;
   1:  PR[91,1] = PR[90,1] + 6.917;
   1:  PR[91,2] = PR[90,2] + 20.554;
   1:L PR[91] R[100]mm/sec CNT100;
   1:  PR[91,1] = PR[90,1] + 6.288;
   1:  PR[91,2] = PR[90,2] + 20.510;
   1:L PR[91] R[100]mm/sec CNT100;
   1:  PR[91,1] = PR[90,1] + 1.780;
   1:  PR[91,2] = PR[90,2] + 19.327;
   1:L PR[91] R[100]mm/sec CNT100;
   1:  PR[91,1] = PR[90,1] + 1.549;
   1:  PR[91,2] = PR[90,2] + 19.260;
   1:L PR[91] R[100]mm/sec CNT100;
   1:  PR[91,1] = PR[90,1] + 1.249;
   1:  PR[91,2] = PR[90,2] + 19.123;
   1:L PR[91] R[100]mm/sec CNT100;
   1:  PR[91,1] = PR[90,1] + 0.347;
   1:  PR[91,2] = PR[90,2] + 18.828;
   1:L PR[91] R[100]mm/sec CNT100;
   1:  PR[91] = PR[90];
   1:  PR[91,1] = PR[90,1] + -0.561;
   1:  PR[91,2] = PR[90,2] + 19.251;
   1:  PR[91,3] = PR[90,3] + 49.595;
   1:L PR[91] R[100]mm/sec CNT100;
   1:  PR[91,1] = PR[90,1] + -1.362;
   1:  PR[91,2] = PR[90,2] + 19.421;
   1:L PR[91] R[100]mm/sec CNT100;
   1:  PR[91,1] = PR[90,1] + -2.914;
   1:  PR[91,2] = PR[90,2] + 19.810;
   1:L PR[91] R[100]mm/sec CNT100;
   1:  PR[91,1] = PR[90,1] + -6.329;
   1:  PR[91,2] = PR[90,2] + 20.706;
   1:L PR[91] R[100]mm/sec CNT100;
   1:  PR[91,1] = PR[90,1] + -6.378;
   1:  PR[91,2] = PR[90,2] + 20.709;
   1:L PR[91] R[100]mm/sec CNT100;
   1:  PR[91,1] = PR[90,1] + -11.149;
   1:  PR[91,2] = PR[90,2] + 20.905;
   1:L PR[91] R[100]mm/sec CNT100;
   1:  PR[91,1] = PR[90,1] + -11.517;
   1:  PR[91,2] = PR[90,2] + 20.852;
   1:L PR[91] R[100]mm/sec CNT100;
   1:  PR[91,1] = PR[90,1] + -15.903;
   1:  PR[91,2] = PR[90,2] + 20.103;
   1:L PR[91] R[100]mm/sec CNT100;
   1:  PR[91,1] = PR[90,1] + -16.554;
   1:  PR[91,2] = PR[90,2] + 19.862;
   1:L PR[91] R[100]mm/sec CNT100;
   1:  PR[91,1] = PR[90,1] + -20.364;
   1:  PR[91,2] = PR[90,2] + 18.343;
   1:L PR[91] R[100]mm/sec CNT100;
   1:  PR[91,1] = PR[90,1] + -21.207;
   1:  PR[91,2] = PR[90,2] + 17.806;
   1:L PR[91] R[100]mm/sec CNT100;
   1:  PR[91,1] = PR[90,1] + -24.323;
   1:  PR[91,2] = PR[90,2] + 15.721;
   1:L PR[91] R[100]mm/sec CNT100;
   1:  PR[91,1] = PR[90,1] + -25.217;
   1:  PR[91,2] = PR[90,2] + 14.831;
   1:L PR[91] R[100]mm/sec CNT100;
   1:  PR[91,1] = PR[90,1] + -27.595;
   1:  PR[91,2] = PR[90,2] + 12.366;
   1:L PR[91] R[100]mm/sec CNT100;
   1:  PR[91,1] = PR[90,1] + -28.383;
   1:  PR[91,2] = PR[90,2] + 11.121;
   1:L PR[91] R[100]mm/sec CNT100;
   1:  PR[91,1] = PR[90,1] + -30.045;
   1:  PR[91,2] = PR[90,2] + 8.409;
   1:L PR[91] R[100]mm/sec CNT100;
   1:  PR[91,1] = PR[90,1] + -30.584;
   1:  PR[91,2] = PR[90,2] + 6.918;
   1:L PR[91] R[100]mm/sec CNT100;
   1:  PR[91,1] = PR[90,1] + -31.552;
   1:  PR[91,2] = PR[90,2] + 4.138;
   1:L PR[91] R[100]mm/sec CNT100;
   1:  PR[91,1] = PR[90,1] + -31.740;
   1:  PR[91,2] = PR[90,2] + 2.488;
   1:L PR[91] R[100]mm/sec CNT100;
   1:  PR[91,1] = PR[90,1] + -31.839;
   1:  PR[91,2] = PR[90,2] + 1.266;
   1:L PR[91] R[100]mm/sec CNT100;
   1:  PR[91,1] = PR[90,1] + -32.028;
   1:  PR[91,2] = PR[90,2] + -0.443;
   1:L PR[91] R[100]mm/sec CNT100;
   1:  PR[91,1] = PR[90,1] + -31.868;
   1:  PR[91,2] = PR[90,2] + -2.137;
   1:L PR[91] R[100]mm/sec CNT100;
   1:  PR[91,1] = PR[90,1] + -31.551;
   1:  PR[91,2] = PR[90,2] + -4.989;
   1:L PR[91] R[100]mm/sec CNT100;
   1:  PR[91,1] = PR[90,1] + -30.584;
   1:  PR[91,2] = PR[90,2] + -7.765;
   1:L PR[91] R[100]mm/sec CNT100;
   1:  PR[91,1] = PR[90,1] + -30.045;
   1:  PR[91,2] = PR[90,2] + -9.256;
   1:L PR[91] R[100]mm/sec CNT100;
   1:  PR[91,1] = PR[90,1] + -28.383;
   1:  PR[91,2] = PR[90,2] + -11.968;
   1:L PR[91] R[100]mm/sec CNT100;
   1:  PR[91,1] = PR[90,1] + -27.595;
   1:  PR[91,2] = PR[90,2] + -13.213;
   1:L PR[91] R[100]mm/sec CNT100;
   1:  PR[91,1] = PR[90,1] + -25.217;
   1:  PR[91,2] = PR[90,2] + -15.678;
   1:L PR[91] R[100]mm/sec CNT100;
   1:  PR[91,1] = PR[90,1] + -24.323;
   1:  PR[91,2] = PR[90,2] + -16.568;
   1:L PR[91] R[100]mm/sec CNT100;
   1:  PR[91,1] = PR[90,1] + -21.207;
   1:  PR[91,2] = PR[90,2] + -18.653;
   1:L PR[91] R[100]mm/sec CNT100;
   1:  PR[91,1] = PR[90,1] + -20.364;
   1:  PR[91,2] = PR[90,2] + -19.190;
   1:L PR[91] R[100]mm/sec CNT100;
   1:  PR[91,1] = PR[90,1] + -16.554;
   1:  PR[91,2] = PR[90,2] + -20.709;
   1:L PR[91] R[100]mm/sec CNT100;
   1:  PR[91,1] = PR[90,1] + -15.902;
   1:  PR[91,2] = PR[90,2] + -20.951;
   1:L PR[91] R[100]mm/sec CNT100;
   1:  PR[91,1] = PR[90,1] + -11.516;
   1:  PR[91,2] = PR[90,2] + -21.700;
   1:L PR[91] R[100]mm/sec CNT100;
   1:  PR[91,1] = PR[90,1] + -11.148;
   1:  PR[91,2] = PR[90,2] + -21.753;
   1:L PR[91] R[100]mm/sec CNT100;
   1:  PR[91,1] = PR[90,1] + -6.377;
   1:  PR[91,2] = PR[90,2] + -21.556;
   1:L PR[91] R[100]mm/sec CNT100;
   1:  PR[91,1] = PR[90,1] + -6.329;
   1:  PR[91,2] = PR[90,2] + -21.553;
   1:L PR[91] R[100]mm/sec CNT100;
   1:  PR[91,1] = PR[90,1] + -2.932;
   1:  PR[91,2] = PR[90,2] + -20.661;
   1:L PR[91] R[100]mm/sec CNT100;
   1:  PR[91,1] = PR[90,1] + -1.282;
   1:  PR[91,2] = PR[90,2] + -20.249;
   1:L PR[91] R[100]mm/sec CNT100;
   1:  PR[91,1] = PR[90,1] + 0.295;
   1:  PR[91,2] = PR[90,2] + -20.024;
   1:L PR[91] R[100]mm/sec CNT100;
   1:  PR[91,1] = PR[90,1] + 1.060;
   1:  PR[91,2] = PR[90,2] + -20.312;
   1:L PR[91] R[100]mm/sec CNT100;
   1:  PR[91,1] = PR[90,1] + 2.450;
   1:  PR[91,2] = PR[90,2] + -20.660;
   1:L PR[91] R[100]mm/sec CNT100;
   1:  PR[91,1] = PR[90,1] + 5.819;
   1:  PR[91,2] = PR[90,2] + -21.545;
   1:L PR[91] R[100]mm/sec CNT100;
   1:  PR[91,1] = PR[90,1] + 10.671;
   1:  PR[91,2] = PR[90,2] + -21.753;
   1:L PR[91] R[100]mm/sec CNT100;
   1:  PR[91,1] = PR[90,1] + 11.037;
   1:  PR[91,2] = PR[90,2] + -21.700;
   1:L PR[91] R[100]mm/sec CNT100;
   1:  PR[91,1] = PR[90,1] + 15.423;
   1:  PR[91,2] = PR[90,2] + -20.950;
   1:L PR[91] R[100]mm/sec CNT100;
   1:  PR[91,1] = PR[90,1] + 16.075;
   1:  PR[91,2] = PR[90,2] + -20.708;
   1:L PR[91] R[100]mm/sec CNT100;
   1:  PR[91,1] = PR[90,1] + 19.885;
   1:  PR[91,2] = PR[90,2] + -19.190;
   1:L PR[91] R[100]mm/sec CNT100;
   1:  PR[91,1] = PR[90,1] + 20.728;
   1:  PR[91,2] = PR[90,2] + -18.654;
   1:L PR[91] R[100]mm/sec CNT100;
   1:  PR[91,1] = PR[90,1] + 23.842;
   1:  PR[91,2] = PR[90,2] + -16.572;
   1:L PR[91] R[100]mm/sec CNT100;
   1:  PR[91,1] = PR[90,1] + 24.735;
   1:  PR[91,2] = PR[90,2] + -15.679;
   1:L PR[91] R[100]mm/sec CNT100;
   1:  PR[91,1] = PR[90,1] + 27.115;
   1:  PR[91,2] = PR[90,2] + -13.208;
   1:L PR[91] R[100]mm/sec CNT100;
   1:  PR[91,1] = PR[90,1] + 27.904;
   1:  PR[91,2] = PR[90,2] + -11.964;
   1:L PR[91] R[100]mm/sec CNT100;
   1:  PR[91,1] = PR[90,1] + 29.566;
   1:  PR[91,2] = PR[90,2] + -9.254;
   1:L PR[91] R[100]mm/sec CNT100;
   1:  PR[91,1] = PR[90,1] + 30.105;
   1:  PR[91,2] = PR[90,2] + -7.770;
   1:L PR[91] R[100]mm/sec CNT100;
   1:  PR[91,1] = PR[90,1] + 31.072;
   1:  PR[91,2] = PR[90,2] + -4.999;
   1:L PR[91] R[100]mm/sec CNT100;
   1:  PR[91,1] = PR[90,1] + 31.260;
   1:  PR[91,2] = PR[90,2] + -3.342;
   1:L PR[91] R[100]mm/sec CNT100;
   1:  PR[91,1] = PR[90,1] + 31.359;
   1:  PR[91,2] = PR[90,2] + -2.117;
   1:L PR[91] R[100]mm/sec CNT100;
   1:  PR[91,1] = PR[90,1] + 31.549;
   1:  PR[91,2] = PR[90,2] + -0.404;
   1:L PR[91] R[100]mm/sec CNT100;
   1:  PR[91,1] = PR[90,1] + 31.388;
   1:  PR[91,2] = PR[90,2] + 1.298;
   1:L PR[91] R[100]mm/sec CNT100;
   1:  PR[91,1] = PR[90,1] + 31.071;
   1:  PR[91,2] = PR[90,2] + 4.154;
   1:L PR[91] R[100]mm/sec CNT100;
   1:  PR[91,1] = PR[90,1] + 30.105;
   1:  PR[91,2] = PR[90,2] + 6.923;
   1:L PR[91] R[100]mm/sec CNT100;
